FUNCTION "TE-ANEI" : VOID	// FC 78
AUTHOR : SIMATIC
FAMILY : EA_DIS
NAME : TE_ANEI
VERSION : 3.0
BEGIN
// (block stored without names or comments; labels and parameter names are numbered)
NETWORK
TITLE =
      L     #PARAM12;
      L     31;
      AW;
      T     MB 200;
      L     #PARAM4;
      T     MW 210;
      A     M 200.0;
      JC    M003;
      L     #PARAM3;
      T     MW 202;
      L     #PARAM1;
      L     W#16#4550;
      ==I;
      JC    M001;
      L     MB 203;
      SLW   3;
      LAR1;
      L     DBW [AR1,P#0.0];
      T     MW 204;
      JU    M002;
M001: NOP   0;
      L     MB 203;
      SLW   3;
      LAR1;
      L     DBW [AR1,P#0.0];
      T     MW 204;
M002: NOP   0;
M003: NOP   0;
NETWORK
TITLE =
      L     MW 210;
      L     2;
      ==I;
      JC    M004;
      JU    M007;
M004: A     M 200.0;
      JC    M008;
      L     MW 204;
      T     MW 240;
      AN    M 240.7;
      JC    M005;
      L     MW 240;
      NEGI;
      DTR;
      L     -1.000000e+00;
      *R;
      JU    M006;
M005: L     MW 240;
      DTR;
M006: T     MD 230;
      L     MD 230;
      L     1.000000e+01;
      /R;
      T     MD 238;
      L     MD 238;
      L     #PARAM7;
      -R;
      T     MD 218;
      L     #PARAM8;
      L     #PARAM7;
      -R;
      T     MD 242;
      L     MD 218;
      L     MD 242;
      /R;
      L     1.000000e+04;
      *R;
      T     MD 214;
      JU    M009;
M007: JU    M011;
M008: JU    M010;
M009: O(;
      L     MD 230;
      L     8.501000e+03;
      >=R;
      );
      O(;
      L     MD 230;
      L     1.000000e+04;
      >=R;
      );
      =     M 240.0;
      O(;
      L     -2.001000e+03;
      L     MD 230;
      >=R;
      );
      O(;
      L     -2.430000e+03;
      L     MD 230;
      >=R;
      );
      =     M 240.1;
      O(;
      L     -2.431000e+03;
      L     MD 230;
      >=R;
      );
      O(;
      L     -3.276800e+04;
      L     MD 230;
      >=R;
      );
      =     M 240.2;
      O(;
      L     MD 230;
      L     1.000000e+04;
      >=R;
      );
      O(;
      L     MD 230;
      L     3.276700e+04;
      >=R;
      );
      =     M 240.3;
      O(;
      L     MD 230;
      L     -2.000000e+03;
      >=R;
      );
      O(;
      L     MD 230;
      L     8.500000e+03;
      >=R;
      );
      =     M 240.4;
      O(;
      A     M 240.0;
      A     M 240.3;
      A     M 240.4;
      );
      O(;
      A     M 240.1;
      A     M 240.2;
      );
      =     M 200.6;
      A     M 200.3;
      A     M 200.6;
      =     M 200.7;
      L     MD 238;
      JU    M012;
M010: R     M 200.7;
      L     #PARAM6;
      T     MD 206;
      L     #PARAM7;
      -R;
      T     MD 244;
      L     #PARAM8;
      L     #PARAM7;
      -R;
      T     MD 248;
      L     MD 244;
      L     MD 248;
      /R;
      L     1.000000e+04;
      *R;
      T     MD 214;
      L     MD 206;
      JU    M014;
M011: JU    M015;
M012: AN    M 200.7;
      ON    M 200.1;
      JC    M013;
      JU    M014;
      L     1.000000e+04;
      T     MD 214;
      L     #PARAM8;
M013: AN    M 200.7;
      ON    M 200.2;
      JC    M014;
      L     0.000000e+00;
      T     MD 214;
      L     #PARAM7;
M014: T     #PARAM10;
      L     MD 214;
      T     #PARAM11;
      L     MB 200;
      T     #PARAM12;
M015: NOP   0;
NETWORK
TITLE =
      L     MW 210;
      L     4;
      ==I;
      JC    M016;
      JU    M020;
M016: A     M 200.0;
      JC    M021;
      L     MW 204;
      T     MW 240;
      AN    M 240.7;
      JC    M018;
M017: L     MW 240;
      NEGI;
      DTR;
      L     -1.000000e+00;
      *R;
      JU    M019;
M018: L     MW 240;
      L     32760;
      >I;
      JC    M017;
      L     MW 240;
      DTR;
M019: T     MD 230;
      L     2.764800e+04;
      /R;
      L     1.000000e+04;
      *R;
      T     MD 214;
      L     #PARAM8;
      L     #PARAM7;
      -R;
      L     1.000000e+04;
      /R;
      T     MD 218;
      L     MD 214;
      L     MD 218;
      *R;
      T     MD 234;
      L     #PARAM7;
      +R;
      T     MD 238;
      JU    M022;
M020: JU    M024;
M021: JU    M023;
M022: O(;
      L     MD 230;
      L     2.764900e+04;
      >=R;
      );
      O(;
      L     MD 230;
      L     3.251100e+04;
      >=R;
      );
      =     M 240.0;
      O(;
      L     -2.764900e+04;
      L     MD 230;
      >=R;
      );
      O(;
      L     -3.251200e+04;
      L     MD 230;
      >=R;
      );
      =     M 240.1;
      O(;
      L     -3.251300e+04;
      L     MD 230;
      >=R;
      );
      O(;
      L     -3.276800e+04;
      L     MD 230;
      >=R;
      );
      =     M 240.2;
      O(;
      L     MD 230;
      L     3.251200e+04;
      >=R;
      );
      O(;
      L     MD 230;
      L     3.276700e+04;
      >=R;
      );
      =     M 240.3;
      O(;
      L     MD 230;
      L     -2.764800e+04;
      >=R;
      );
      O(;
      L     MD 230;
      L     2.764800e+04;
      >=R;
      );
      =     M 240.4;
      O(;
      A     M 240.0;
      A     M 240.3;
      A     M 240.4;
      );
      O(;
      A     M 240.1;
      A     M 240.2;
      );
      =     M 200.6;
      A     M 200.3;
      A     M 200.6;
      =     M 200.7;
      L     MD 238;
      JU    M025;
M023: R     M 200.7;
      L     #PARAM6;
      T     MD 206;
      L     #PARAM7;
      -R;
      T     MD 244;
      L     #PARAM8;
      L     #PARAM7;
      -R;
      T     MD 248;
      L     MD 244;
      L     MD 248;
      /R;
      L     1.000000e+04;
      *R;
      T     MD 214;
      L     MD 206;
      JU    M027;
M024: JU    M028;
M025: AN    M 200.7;
      ON    M 200.1;
      JC    M026;
      JU    M027;
      L     1.000000e+04;
      T     MD 214;
      L     #PARAM8;
M026: AN    M 200.7;
      ON    M 200.2;
      JC    M027;
      L     0.000000e+00;
      T     MD 214;
      L     #PARAM7;
M027: T     #PARAM10;
      L     MD 214;
      T     #PARAM11;
      L     MB 200;
      T     #PARAM12;
M028: NOP   0;
NETWORK
TITLE =
      L     MW 210;
      L     6;
      ==I;
      JC    M029;
      JU    M033;
M029: A     M 200.0;
      JC    M034;
      L     MW 204;
      T     MW 240;
      AN    M 240.7;
      JC    M031;
M030: L     MW 240;
      NEGI;
      DTR;
      L     -1.000000e+00;
      *R;
      JU    M032;
M031: L     MW 240;
      L     32760;
      >I;
      JC    M030;
      L     MW 240;
      DTR;
M032: T     MD 230;
      L     2.764800e+04;
      /R;
      L     1.000000e+04;
      *R;
      T     MD 214;
      L     #PARAM8;
      L     #PARAM7;
      -R;
      L     1.000000e+04;
      /R;
      T     MD 218;
      L     MD 214;
      L     MD 218;
      *R;
      T     MD 234;
      L     #PARAM7;
      +R;
      T     MD 238;
      JU    M035;
M033: JU    M037;
M034: JU    M036;
M035: O(;
      L     MD 230;
      L     2.764900e+04;
      >=R;
      );
      O(;
      L     MD 230;
      L     3.251100e+04;
      >=R;
      );
      =     M 240.0;
      O(;
      L     -1.000000e+00;
      L     MD 230;
      >=R;
      );
      O(;
      L     -4.864000e+03;
      L     MD 230;
      >=R;
      );
      =     M 240.1;
      O(;
      L     -4.865000e+03;
      L     MD 230;
      >=R;
      );
      O(;
      L     -3.276800e+04;
      L     MD 230;
      >=R;
      );
      =     M 240.2;
      O(;
      L     MD 230;
      L     3.251200e+04;
      >=R;
      );
      O(;
      L     MD 230;
      L     3.276700e+04;
      >=R;
      );
      =     M 240.3;
      O(;
      L     MD 230;
      L     0.000000e+00;
      >=R;
      );
      O(;
      L     MD 230;
      L     2.764800e+04;
      >=R;
      );
      =     M 240.4;
      O(;
      A     M 240.0;
      A     M 240.3;
      A     M 240.4;
      );
      O(;
      A     M 240.1;
      A     M 240.2;
      );
      =     M 200.6;
      A     M 200.3;
      A     M 200.6;
      =     M 200.7;
      L     MD 238;
      JU    M038;
M036: R     M 200.7;
      L     #PARAM6;
      T     MD 206;
      L     #PARAM7;
      -R;
      T     MD 244;
      L     #PARAM8;
      L     #PARAM7;
      -R;
      T     MD 248;
      L     MD 244;
      L     MD 248;
      /R;
      L     1.000000e+04;
      *R;
      T     MD 214;
      L     MD 206;
      JU    M040;
M037: JU    M041;
M038: AN    M 200.7;
      ON    M 200.1;
      JC    M039;
      JU    M040;
      L     1.000000e+04;
      T     MD 214;
      L     #PARAM8;
M039: AN    M 200.7;
      ON    M 200.2;
      JC    M040;
      L     0.000000e+00;
      T     MD 214;
      L     #PARAM7;
M040: T     #PARAM10;
      L     MD 214;
      T     #PARAM11;
      L     MB 200;
      T     #PARAM12;
M041: NOP   0;
NETWORK
TITLE =
      L     MW 210;
      L     7;
      ==I;
      JC    M042;
      JU    M046;
M042: A     M 200.0;
      JC    M047;
      L     MW 204;
      T     MW 240;
      AN    M 240.7;
      JC    M044;
M043: L     MW 240;
      NEGI;
      DTR;
      L     -1.000000e+00;
      *R;
      JU    M045;
M044: L     MW 240;
      L     32760;
      >I;
      JC    M043;
      L     MW 240;
      DTR;
M045: T     MD 230;
      L     1.820000e+04;
      /R;
      L     1.000000e+04;
      *R;
      T     MD 214;
      L     #PARAM8;
      L     #PARAM7;
      -R;
      L     1.000000e+04;
      /R;
      T     MD 218;
      L     MD 214;
      L     MD 218;
      *R;
      T     MD 234;
      L     #PARAM7;
      +R;
      T     MD 238;
      JU    M048;
M046: JU    M050;
M047: JU    M049;
M048: O(;
      L     MD 230;
      L     1.820100e+04;
      >=R;
      );
      O(;
      L     MD 230;
      L     2.070000e+04;
      >=R;
      );
      =     M 240.0;
      O(;
      L     -1.000000e+00;
      L     MD 230;
      >=R;
      );
      O(;
      L     -1.200000e+03;
      L     MD 230;
      >=R;
      );
      =     M 240.1;
      L     -3.276800e+04;
      L     MD 230;
      >=R;
      =     M 240.2;
      L     MD 230;
      L     2.070100e+04;
      >=R;
      =     M 240.3;
      O(;
      L     MD 230;
      L     0.000000e+00;
      >=R;
      );
      O(;
      L     MD 230;
      L     1.820000e+04;
      >=R;
      );
      =     M 240.4;
      O(;
      A     M 240.0;
      A     M 240.3;
      A     M 240.4;
      );
      O(;
      A     M 240.1;
      A     M 240.2;
      );
      =     M 200.6;
      A     M 200.3;
      A     M 200.6;
      =     M 200.7;
      L     MD 238;
      JU    M051;
M049: R     M 200.7;
      L     #PARAM6;
      T     MD 206;
      L     #PARAM7;
      -R;
      T     MD 244;
      L     #PARAM8;
      L     #PARAM7;
      -R;
      T     MD 248;
      L     MD 244;
      L     MD 248;
      /R;
      L     1.000000e+04;
      *R;
      T     MD 214;
      L     MD 206;
      JU    M053;
M050: JU    M054;
M051: AN    M 200.7;
      ON    M 200.1;
      JC    M052;
      JU    M053;
      L     1.000000e+04;
      T     MD 214;
      L     #PARAM8;
M052: AN    M 200.7;
      ON    M 200.2;
      JC    M053;
      L     0.000000e+00;
      T     MD 214;
      L     #PARAM7;
M053: T     #PARAM10;
      L     MD 214;
      T     #PARAM11;
      L     MB 200;
      T     #PARAM12;
M054: NOP   0;
NETWORK
TITLE =
      L     MW 210;
      L     8;
      ==I;
      JC    M055;
      JU    M059;
M055: A     M 200.0;
      JC    M060;
      L     MW 204;
      T     MW 240;
      AN    M 240.7;
      JC    M057;
M056: L     MW 240;
      NEGI;
      DTR;
      L     -1.000000e+00;
      *R;
      JU    M058;
M057: L     MW 240;
      L     32760;
      >I;
      JC    M056;
      L     MW 240;
      DTR;
M058: T     MD 230;
      L     2.315000e+04;
      /R;
      L     1.000000e+04;
      *R;
      T     MD 214;
      L     #PARAM8;
      L     #PARAM7;
      -R;
      L     1.000000e+04;
      /R;
      T     MD 218;
      L     MD 214;
      L     MD 218;
      *R;
      T     MD 234;
      L     #PARAM7;
      +R;
      T     MD 238;
      JU    M061;
M059: JU    M063;
M060: JU    M062;
M061: O(;
      L     MD 230;
      L     2.500000e+04;
      >=R;
      );
      O(;
      L     MD 230;
      L     2.315100e+04;
      >=R;
      );
      =     M 240.0;
      O(;
      L     -1.000000e+00;
      L     MD 230;
      >=R;
      );
      O(;
      L     -1.200000e+03;
      L     MD 230;
      >=R;
      );
      =     M 240.1;
      L     -3.276800e+04;
      L     MD 230;
      >=R;
      =     M 240.2;
      L     MD 230;
      L     2.500100e+04;
      >=R;
      =     M 240.3;
      O(;
      L     MD 230;
      L     0.000000e+00;
      >=R;
      );
      O(;
      L     MD 230;
      L     2.315000e+04;
      >=R;
      );
      =     M 240.4;
      O(;
      A     M 240.0;
      A     M 240.3;
      A     M 240.4;
      );
      O(;
      A     M 240.1;
      A     M 240.2;
      );
      =     M 200.6;
      A     M 200.3;
      A     M 200.6;
      =     M 200.7;
      L     MD 238;
      JU    M064;
M062: R     M 200.7;
      L     #PARAM6;
      T     MD 206;
      L     #PARAM7;
      -R;
      T     MD 244;
      L     #PARAM8;
      L     #PARAM7;
      -R;
      T     MD 248;
      L     MD 244;
      L     MD 248;
      /R;
      L     1.000000e+04;
      *R;
      T     MD 214;
      L     MD 206;
      JU    M066;
M063: JU    M067;
M064: AN    M 200.7;
      ON    M 200.1;
      JC    M065;
      JU    M066;
      L     1.000000e+04;
      T     MD 214;
      L     #PARAM8;
M065: AN    M 200.7;
      ON    M 200.2;
      JC    M066;
      L     0.000000e+00;
      T     MD 214;
      L     #PARAM7;
M066: T     #PARAM10;
      L     MD 214;
      T     #PARAM11;
      L     MB 200;
      T     #PARAM12;
M067: NOP   0;
NETWORK
TITLE =
      L     MW 210;
      L     9;
      ==I;
      JC    M068;
      JU    M073;
M068: A     M 200.0;
      JC    M074;
      L     MW 204;
      T     MW 240;
      AN    M 240.7;
      JC    M070;
M069: L     MW 240;
      NEGI;
      DTR;
      L     -1.000000e+00;
      *R;
      JU    M071;
M070: L     MW 240;
      L     32760;
      >I;
      JC    M069;
      L     MW 240;
      DTR;
      JU    M072;
M071: T     MD 230;
      L     #PARAM7;
      L     1.000000e+01;
      *R;
      T     MD 242;
      L     MD 230;
      L     MD 242;
      -R;
      L     1.270000e+04;
      /R;
      L     1.000000e+04;
      *R;
      T     MD 214;
      L     #PARAM8;
      L     #PARAM7;
      -R;
      L     1.000000e+04;
      /R;
      T     MD 218;
      L     MD 214;
      L     MD 218;
      *R;
      T     MD 234;
      L     #PARAM7;
      +R;
      T     MD 238;
      JU    M075;
M072: T     MD 230;
      L     #PARAM7;
      L     -1.000000e+01;
      *R;
      T     MD 242;
      L     MD 230;
      L     MD 242;
      +R;
      L     1.270000e+04;
      /R;
      L     1.000000e+04;
      *R;
      T     MD 214;
      L     #PARAM8;
      L     #PARAM7;
      -R;
      L     1.000000e+04;
      /R;
      T     MD 218;
      L     MD 214;
      L     MD 218;
      *R;
      T     MD 234;
      L     #PARAM7;
      +R;
      T     MD 238;
      JU    M075;
M073: JU    M077;
M074: JU    M076;
M075: O(;
      L     MD 230;
      L     1.200000e+04;
      >=R;
      );
      O(;
      L     MD 230;
      L     1.000100e+04;
      >=R;
      );
      =     M 240.0;
      O(;
      L     -1.000000e+00;
      L     MD 230;
      >=R;
      );
      O(;
      L     -1.200000e+03;
      L     MD 230;
      >=R;
      );
      =     M 240.1;
      L     -3.276800e+04;
      L     MD 230;
      >=R;
      =     M 240.2;
      L     MD 230;
      L     2.500100e+04;
      >=R;
      =     M 240.3;
      O(;
      L     MD 230;
      L     -2.700000e+03;
      >=R;
      );
      O(;
      L     MD 230;
      L     1.000000e+04;
      >=R;
      );
      =     M 240.4;
      O(;
      A     M 240.0;
      A     M 240.3;
      A     M 240.4;
      );
      O(;
      A     M 240.1;
      A     M 240.2;
      );
      =     M 200.6;
      A     M 200.3;
      A     M 200.6;
      =     M 200.7;
      L     MD 238;
      JU    M078;
M076: R     M 200.7;
      L     #PARAM6;
      T     MD 206;
      L     #PARAM7;
      -R;
      T     MD 244;
      L     #PARAM8;
      L     #PARAM7;
      -R;
      T     MD 248;
      L     MD 244;
      L     MD 248;
      /R;
      L     1.000000e+04;
      *R;
      T     MD 214;
      L     MD 206;
      JU    M080;
M077: JU    M081;
M078: AN    M 200.7;
      ON    M 200.1;
      JC    M079;
      JU    M080;
      L     1.000000e+04;
      T     MD 214;
      L     #PARAM8;
M079: AN    M 200.7;
      ON    M 200.2;
      JC    M040;
      L     0.000000e+00;
      T     MD 214;
      L     #PARAM7;
M080: T     #PARAM10;
      L     MD 214;
      T     #PARAM11;
      L     MB 200;
      T     #PARAM12;
M081: NOP   0;
NETWORK
TITLE =
      L     MW 210;
      L     10;
      ==I;
      JC    M082;
      JU    M085;
M082: A     M 200.0;
      JC    M086;
      L     MW 204;
      T     MW 240;
      AN    M 240.7;
      JC    M083;
      L     MW 240;
      NEGI;
      DTR;
      L     -1.000000e+00;
      *R;
      JU    M084;
M083: L     MW 240;
      DTR;
M084: T     MD 230;
      L     MD 230;
      L     1.000000e+01;
      /R;
      T     MD 238;
      L     MD 238;
      L     #PARAM7;
      -R;
      T     MD 218;
      L     #PARAM8;
      L     #PARAM7;
      -R;
      T     MD 242;
      L     MD 218;
      L     MD 242;
      /R;
      L     1.000000e+04;
      *R;
      T     MD 214;
      JU    M087;
M085: JU    M089;
M086: JU    M088;
M087: O(;
      L     MD 230;
      L     1.200100e+04;
      >=R;
      );
      O(;
      L     MD 230;
      L     1.450000e+04;
      >=R;
      );
      =     M 240.0;
      L     -2.100000e+03;
      L     MD 230;
      >=R;
      =     M 240.1;
      L     -2.100000e+03;
      L     MD 230;
      >=R;
      =     M 240.2;
      L     MD 230;
      L     1.450100e+04;
      >=R;
      =     M 240.3;
      O(;
      L     MD 230;
      L     -2.100000e+03;
      >=R;
      );
      O(;
      L     MD 230;
      L     1.200000e+03;
      >=R;
      );
      =     M 240.4;
      O(;
      A     M 240.0;
      A     M 240.3;
      A     M 240.4;
      );
      O(;
      A     M 240.1;
      A     M 240.2;
      );
      =     M 200.6;
      A     M 200.3;
      A     M 200.6;
      =     M 200.7;
      L     MD 238;
      JU    M090;
M088: R     M 200.7;
      L     #PARAM6;
      T     MD 206;
      L     #PARAM7;
      -R;
      T     MD 244;
      L     #PARAM8;
      L     #PARAM7;
      -R;
      T     MD 248;
      L     MD 244;
      L     MD 248;
      /R;
      L     1.000000e+04;
      *R;
      T     MD 214;
      L     MD 206;
      JU    M092;
M089: JU    M093;
M090: AN    M 200.7;
      ON    M 200.1;
      JC    M091;
      JU    M092;
      L     1.000000e+04;
      T     MD 214;
      L     #PARAM8;
M091: AN    M 200.7;
      ON    M 200.2;
      JC    M092;
      L     0.000000e+00;
      T     MD 214;
      L     #PARAM7;
M092: T     #PARAM10;
      L     MD 214;
      T     #PARAM11;
      L     MB 200;
      T     #PARAM12;
M093: NOP   0;
NETWORK
TITLE =
      L     MW 210;
      L     11;
      ==I;
      JC    M094;
      JU    M097;
M094: A     M 200.0;
      JC    M098;
      L     MW 204;
      T     MW 240;
      AN    M 240.7;
      JC    M095;
      L     MW 240;
      NEGI;
      DTR;
      L     -1.000000e+00;
      *R;
      JU    M096;
M095: L     MW 240;
      DTR;
M096: T     MD 230;
      L     MD 230;
      L     1.000000e+01;
      /R;
      T     MD 238;
      L     MD 238;
      L     #PARAM7;
      -R;
      T     MD 218;
      L     #PARAM8;
      L     #PARAM7;
      -R;
      T     MD 242;
      L     MD 218;
      L     MD 242;
      /R;
      L     1.000000e+04;
      *R;
      T     MD 214;
      JU    M099;
M097: JU    M101;
M098: JU    M100;
M099: O(;
      L     MD 230;
      L     1.666200e+04;
      >=R;
      );
      O(;
      L     MD 230;
      L     1.372100e+04;
      >=R;
      );
      =     M 240.0;
      L     -2.700000e+03;
      L     MD 230;
      >=R;
      =     M 240.1;
      L     -2.700000e+03;
      L     MD 230;
      >=R;
      =     M 240.2;
      L     MD 230;
      L     1.622100e+04;
      >=R;
      =     M 240.3;
      O(;
      L     MD 230;
      L     -2.700000e+03;
      >=R;
      );
      O(;
      L     MD 230;
      L     1.372000e+03;
      >=R;
      );
      =     M 240.4;
      O(;
      A     M 240.0;
      A     M 240.3;
      A     M 240.4;
      );
      O(;
      A     M 240.1;
      A     M 240.2;
      );
      =     M 200.6;
      A     M 200.3;
      A     M 200.6;
      =     M 200.7;
      L     MD 238;
      JU    M102;
M100: R     M 200.7;
      L     #PARAM6;
      T     MD 206;
      L     #PARAM7;
      -R;
      T     MD 244;
      L     #PARAM8;
      L     #PARAM7;
      -R;
      T     MD 248;
      L     MD 244;
      L     MD 248;
      /R;
      L     1.000000e+04;
      *R;
      T     MD 214;
      L     MD 206;
      JU    M104;
M101: JU    M105;
M102: AN    M 200.7;
      ON    M 200.1;
      JC    M103;
      JU    M104;
      L     1.000000e+04;
      T     MD 214;
      L     #PARAM8;
M103: AN    M 200.7;
      ON    M 200.2;
      JC    M104;
      L     0.000000e+00;
      T     MD 214;
      L     #PARAM7;
M104: T     #PARAM10;
      L     MD 214;
      T     #PARAM11;
      L     MB 200;
      T     #PARAM12;
M105: NOP   0;
NETWORK
TITLE =
      L     MW 210;
      L     12;
      ==I;
      JC    M106;
      JU    M109;
M106: A     M 200.0;
      JC    M110;
      L     MW 204;
      T     MW 240;
      AN    M 240.7;
      JC    M107;
      L     MW 240;
      NEGI;
      DTR;
      L     -1.000000e+00;
      *R;
      JU    M108;
M107: L     MW 240;
      DTR;
M108: T     MD 230;
      L     MD 230;
      L     1.000000e+01;
      /R;
      T     MD 238;
      L     MD 238;
      L     #PARAM7;
      -R;
      T     MD 218;
      L     #PARAM8;
      L     #PARAM7;
      -R;
      T     MD 242;
      L     MD 218;
      L     MD 242;
      /R;
      L     1.000000e+04;
      *R;
      T     MD 214;
      JU    M111;
M109: JU    M113;
M110: JU    M112;
M111: O(;
      L     MD 230;
      L     1.150000e+04;
      >=R;
      );
      O(;
      L     MD 230;
      L     9.001000e+03;
      >=R;
      );
      =     M 240.0;
      L     -2.000000e+03;
      L     MD 230;
      >=R;
      =     M 240.1;
      L     -2.000000e+03;
      L     MD 230;
      >=R;
      =     M 240.2;
      L     MD 230;
      L     9.001000e+03;
      >=R;
      =     M 240.3;
      O(;
      L     MD 230;
      L     -2.000000e+03;
      >=R;
      );
      O(;
      L     MD 230;
      L     9.000000e+03;
      >=R;
      );
      =     M 240.4;
      O(;
      A     M 240.0;
      A     M 240.3;
      A     M 240.4;
      );
      O(;
      A     M 240.1;
      A     M 240.2;
      );
      =     M 200.6;
      A     M 200.3;
      A     M 200.6;
      =     M 200.7;
      L     MD 238;
      JU    M114;
M112: R     M 200.7;
      L     #PARAM6;
      T     MD 206;
      L     #PARAM7;
      -R;
      T     MD 244;
      L     #PARAM8;
      L     #PARAM7;
      -R;
      T     MD 248;
      L     MD 244;
      L     MD 248;
      /R;
      L     1.000000e+04;
      *R;
      T     MD 214;
      L     MD 206;
      JU    M116;
M113: JU    M117;
M114: AN    M 200.7;
      ON    M 200.1;
      JC    M115;
      JU    M116;
      L     1.000000e+04;
      T     MD 214;
      L     #PARAM8;
M115: AN    M 200.7;
      ON    M 200.2;
      JC    M116;
      L     0.000000e+00;
      T     MD 214;
      L     #PARAM7;
M116: T     #PARAM10;
      L     MD 214;
      T     #PARAM11;
      L     MB 200;
      T     #PARAM12;
M117: NOP   0;
NETWORK
TITLE =
      L     MW 210;
      L     12;
      ==I;
      JC    M118;
      JU    M121;
M118: A     M 200.0;
      JC    M122;
      L     MW 204;
      T     MW 240;
      AN    M 240.7;
      JC    M119;
      L     MW 240;
      NEGI;
      DTR;
      L     -1.000000e+00;
      *R;
      JU    M120;
M119: L     MW 240;
      DTR;
M120: T     MD 230;
      L     MD 230;
      L     1.000000e+01;
      /R;
      T     MD 238;
      L     MD 238;
      L     #PARAM7;
      -R;
      T     MD 218;
      L     #PARAM8;
      L     #PARAM7;
      -R;
      T     MD 242;
      L     MD 218;
      L     MD 242;
      /R;
      L     1.000000e+04;
      *R;
      T     MD 214;
      JU    M123;
M121: JU    M125;
M122: JU    M124;
M123: O(;
      L     MD 230;
      L     1.550000e+04;
      >=R;
      );
      O(;
      L     MD 230;
      L     1.300100e+04;
      >=R;
      );
      =     M 240.0;
      L     -2.700000e+03;
      L     MD 230;
      >=R;
      =     M 240.1;
      L     -2.700000e+03;
      L     MD 230;
      >=R;
      =     M 240.2;
      L     MD 230;
      L     1.550100e+04;
      >=R;
      =     M 240.3;
      O(;
      L     MD 230;
      L     -2.700000e+03;
      >=R;
      );
      O(;
      L     MD 230;
      L     1.550000e+03;
      >=R;
      );
      =     M 240.4;
      O(;
      A     M 240.0;
      A     M 240.3;
      A     M 240.4;
      );
      O(;
      A     M 240.1;
      A     M 240.2;
      );
      =     M 200.6;
      A     M 200.3;
      A     M 200.6;
      =     M 200.7;
      L     MD 238;
      JU    M126;
M124: R     M 200.7;
      L     #PARAM6;
      T     MD 206;
      L     #PARAM7;
      -R;
      T     MD 244;
      L     #PARAM8;
      L     #PARAM7;
      -R;
      T     MD 248;
      L     MD 244;
      L     MD 248;
      /R;
      L     1.000000e+04;
      *R;
      T     MD 214;
      L     MD 206;
      JU    M128;
M125: JU    M129;
M126: AN    M 200.7;
      ON    M 200.1;
      JC    M127;
      JU    M128;
      L     1.000000e+04;
      T     MD 214;
      L     #PARAM8;
M127: AN    M 200.7;
      ON    M 200.2;
      JC    M128;
      L     0.000000e+00;
      T     MD 214;
      L     #PARAM7;
M128: T     #PARAM10;
      L     MD 214;
      T     #PARAM11;
      L     MB 200;
      T     #PARAM12;
M129: NOP   0;
NETWORK
TITLE =
      L     MW 210;
      L     14;
      ==I;
      JC    M130;
      JU    M133;
M130: A     M 200.0;
      JC    M134;
      L     MW 204;
      T     MW 240;
      AN    M 240.7;
      JC    M131;
      L     MW 240;
      NEGI;
      DTR;
      L     -1.000000e+00;
      *R;
      JU    M132;
M131: L     MW 240;
      DTR;
M132: T     MD 230;
      L     MD 230;
      L     1.000000e+01;
      /R;
      T     MD 238;
      L     MD 238;
      L     #PARAM7;
      -R;
      T     MD 218;
      L     #PARAM8;
      L     #PARAM7;
      -R;
      T     MD 242;
      L     MD 218;
      L     MD 242;
      /R;
      L     1.000000e+04;
      *R;
      T     MD 214;
      JU    M135;
M133: JU    M137;
M134: JU    M136;
M135: O(;
      L     MD 230;
      L     2.019000e+04;
      >=R;
      );
      O(;
      L     MD 230;
      L     1.769100e+04;
      >=R;
      );
      =     M 240.0;
      O(;
      L     -5.010000e+02;
      L     MD 230;
      >=R;
      );
      O(;
      L     -1.700000e+03;
      L     MD 230;
      >=R;
      );
      =     M 240.1;
      O(;
      L     2.090100e+04;
      L     MD 230;
      >=R;
      );
      O(;
      L     -1.200000e+03;
      L     MD 230;
      >=R;
      );
      =     M 240.2;
      O(;
      L     -1.000000e+00;
      L     MD 230;
      >=R;
      );
      O(;
      L     -1.200000e+03;
      L     MD 230;
      >=R;
      );
      =     M 240.3;
      O(;
      L     MD 230;
      L     -5.000000e+02;
      >=R;
      );
      O(;
      L     MD 230;
      L     1.769000e+04;
      >=R;
      );
      =     M 240.4;
      O(;
      A     M 240.0;
      A     M 240.3;
      A     M 240.4;
      );
      O(;
      A     M 240.1;
      A     M 240.2;
      );
      =     M 200.6;
      A     M 200.3;
      A     M 200.6;
      =     M 200.7;
      L     MD 238;
      JU    M138;
M136: R     M 200.7;
      L     #PARAM6;
      T     MD 206;
      L     #PARAM7;
      -R;
      T     MD 244;
      L     #PARAM8;
      L     #PARAM7;
      -R;
      T     MD 248;
      L     MD 244;
      L     MD 248;
      /R;
      L     1.000000e+04;
      *R;
      T     MD 214;
      L     MD 206;
      JU    M140;
M137: JU    M141;
M138: AN    M 200.7;
      ON    M 200.1;
      JC    M139;
      JU    M140;
      L     1.000000e+04;
      T     MD 214;
      L     #PARAM8;
M139: AN    M 200.7;
      ON    M 200.2;
      JC    M140;
      L     0.000000e+00;
      T     MD 214;
      L     #PARAM7;
M140: T     #PARAM10;
      L     MD 214;
      T     #PARAM11;
      L     MB 200;
      T     #PARAM12;
M141: NOP   0;
NETWORK
TITLE =
      L     MW 210;
      L     14;
      ==I;
      JC    M142;
      JU    M145;
M142: A     M 200.0;
      JC    M146;
      L     MW 204;
      T     MW 240;
      AN    M 240.7;
      JC    M143;
      L     MW 240;
      NEGI;
      DTR;
      L     -1.000000e+00;
      *R;
      JU    M144;
M143: L     MW 240;
      DTR;
M144: T     MD 230;
      L     MD 230;
      L     1.000000e+01;
      /R;
      T     MD 238;
      L     MD 238;
      L     #PARAM7;
      -R;
      T     MD 218;
      L     #PARAM8;
      L     #PARAM7;
      -R;
      T     MD 242;
      L     MD 218;
      L     MD 242;
      /R;
      L     1.000000e+04;
      *R;
      T     MD 214;
      JU    M147;
M145: JU    M149;
M146: JU    M148;
M147: O(;
      L     MD 230;
      L     1.666200e+04;
      >=R;
      );
      O(;
      L     MD 230;
      L     1.372100e+04;
      >=R;
      );
      =     M 240.0;
      L     -2.700000e+03;
      L     MD 230;
      >=R;
      =     M 240.1;
      L     -2.700000e+03;
      L     MD 230;
      >=R;
      =     M 240.2;
      L     MD 230;
      L     1.622100e+04;
      >=R;
      =     M 240.3;
      O(;
      L     MD 230;
      L     -2.700000e+03;
      >=R;
      );
      O(;
      L     MD 230;
      L     1.372000e+03;
      >=R;
      );
      =     M 240.4;
      O(;
      A     M 240.0;
      A     M 240.3;
      A     M 240.4;
      );
      O(;
      A     M 240.1;
      A     M 240.2;
      );
      =     M 200.6;
      A     M 200.3;
      A     M 200.6;
      =     M 200.7;
      L     MD 238;
      JU    M150;
M148: R     M 200.7;
      L     #PARAM6;
      T     MD 206;
      L     #PARAM7;
      -R;
      T     MD 244;
      L     #PARAM8;
      L     #PARAM7;
      -R;
      T     MD 248;
      L     MD 244;
      L     MD 248;
      /R;
      L     1.000000e+04;
      *R;
      T     MD 214;
      L     MD 206;
      JU    M152;
M149: JU    M153;
M150: AN    M 200.7;
      ON    M 200.1;
      JC    M151;
      JU    M152;
      L     1.000000e+04;
      T     MD 214;
      L     #PARAM8;
M151: AN    M 200.7;
      ON    M 200.2;
      JC    M152;
      L     0.000000e+00;
      T     MD 214;
      L     #PARAM7;
M152: T     #PARAM10;
      L     MD 214;
      T     #PARAM11;
      L     MB 200;
      T     #PARAM12;
M153: NOP   0;
NETWORK
TITLE =
      L     0;
      L     #PARAM9;
      ==I;
      BEC;
      T     MW 206;
      T     MW 220;
      L     MB 206;
      SLW   3;
      LAR1;
      L     DBW [AR1,P#0.0];
      T     MW 208;
      L     MW 220;
      SLW   12;
      SRW   12;
      T     MW 220;
      L     8;
      L     MB 221;
      >I;
      JC    M154;
      +     -8;
      SLW   8;
      INC   208;
      JU    M155;
M154: SLW   8;
      INC   209;
M155: T     MW 210;
      L     MB 210;
      L     MB 211;
      SLW   3;
      OW;
      LAR2;
      A     M 200.7;
      =     M [AR2,P#0.0];
      L     MB 206;
      SLW   3;
      LAR1;
      L     MW 208;
      T     DBW [AR1,P#0.0];
END_FUNCTION

FUNCTION "TE-ANAU" : VOID	// FC 79
AUTHOR : SIMATIC
FAMILY : EA_DIS
NAME : TE_ANAU
VERSION : 3.0
BEGIN
// (block stored without names or comments; labels and parameter names are numbered)
NETWORK
TITLE =
      L     #PARAM1;
      T     MB 255;
      L     #PARAM3;
      T     MB 254;
      L     1;
      >I;
      JC    M001;
      L     #PARAM2;
      L     2.764800e+00;
      *R;
      RND;
      T     MW 240;
      JU    M004;
M001: L     #PARAM2;
      L     0.000000e+00;
      <R;
      JC    M002;
      TAK;
      L     2.764800e+00;
      *R;
      T     MD 250;
      JU    M003;
M002: TAK;
      L     -1.000000e+00;
      *R;
M003: RND;
      T     MW 240;
M004: A     M 255.1;
      JC    M005;
      L     MW 240;
      T     #PARAM4;
M005: NOP   0;
END_FUNCTION

FUNCTION "FC 110" : VOID	// FC 110
VERSION : 0.1
BEGIN
// (block stored without names or comments; labels and parameter names are numbered)
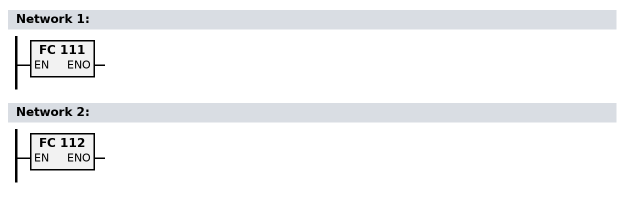
NETWORK
TITLE =
      CALL  "FC 111";
      NOP   0;
NETWORK
TITLE =
      CALL  "FC 112";
      NOP   0;
END_FUNCTION

FUNCTION "FC 111" : VOID	// FC 111
VERSION : 0.1
BEGIN
// (block stored without names or comments; labels and parameter names are numbered)
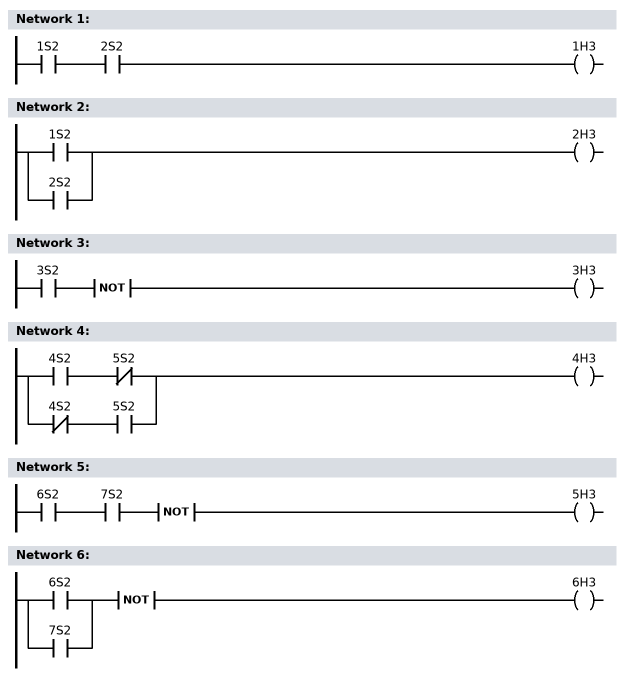
NETWORK
TITLE =
      A     "1S2";
      A     "2S2";
      =     "1H3";
NETWORK
TITLE =
      O     "1S2";
      O     "2S2";
      =     "2H3";
NETWORK
TITLE =
      A     "3S2";
      NOT;
      =     "3H3";
NETWORK
TITLE =
      A     "4S2";
      AN    "5S2";
      O;
      AN    "4S2";
      A     "5S2";
      =     "4H3";
NETWORK
TITLE =
      A     "6S2";
      A     "7S2";
      NOT;
      =     "5H3";
NETWORK
TITLE =
      A(;
      O     "6S2";
      O     "7S2";
      );
      NOT;
      =     "6H3";
END_FUNCTION

FUNCTION "FC 112" : VOID	// FC 112
VERSION : 0.1
BEGIN
// (block stored without names or comments; labels and parameter names are numbered)
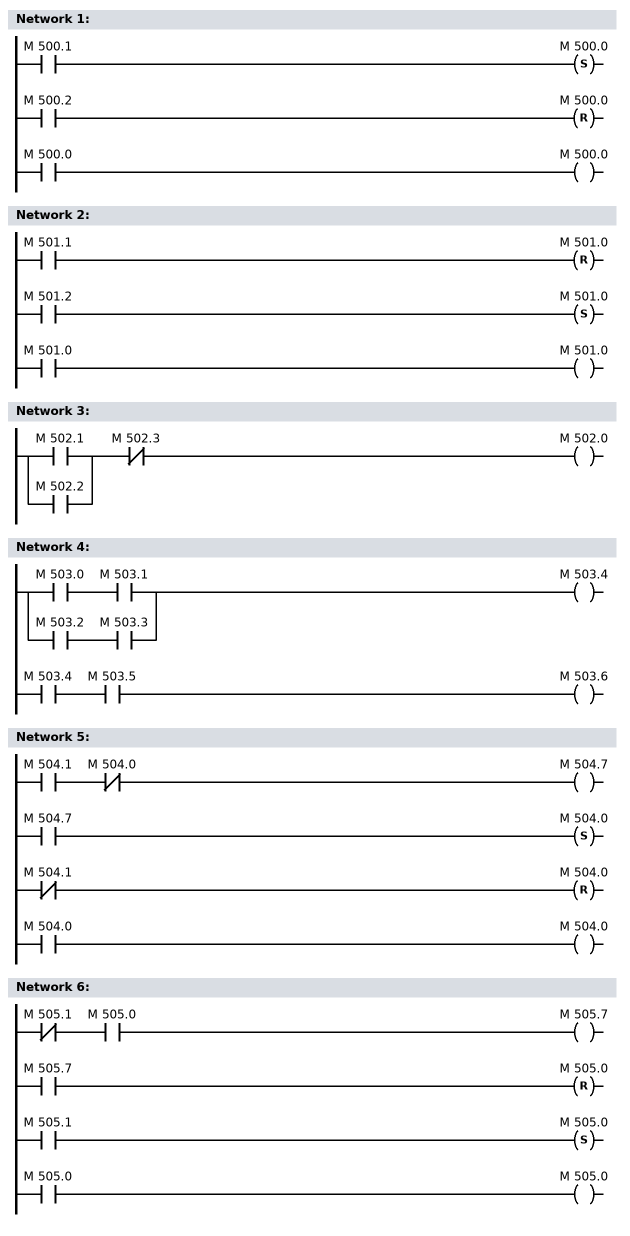
NETWORK
TITLE =
      A     M 500.1;
      S     M 500.0;
      A     M 500.2;
      R     M 500.0;
      A     M 500.0;
      =     M 500.0;
NETWORK
TITLE =
      A     M 501.1;
      R     M 501.0;
      A     M 501.2;
      S     M 501.0;
      A     M 501.0;
      =     M 501.0;
NETWORK
TITLE =
      A(;
      O     M 502.1;
      O     M 502.2;
      );
      AN    M 502.3;
      =     M 502.0;
NETWORK
TITLE =
      A(;
      A     M 503.0;
      A     M 503.1;
      O;
      A     M 503.2;
      A     M 503.3;
      );
      =     M 503.4;
      A     M 503.4;
      A     M 503.5;
      =     M 503.6;
NETWORK
TITLE =
      A     M 504.1;
      AN    M 504.0;
      =     M 504.7;
      A     M 504.7;
      S     M 504.0;
      AN    M 504.1;
      R     M 504.0;
      A     M 504.0;
      =     M 504.0;
NETWORK
TITLE =
      AN    M 505.1;
      A     M 505.0;
      =     M 505.7;
      A     M 505.7;
      R     M 505.0;
      A     M 505.1;
      S     M 505.0;
      A     M 505.0;
      =     M 505.0;
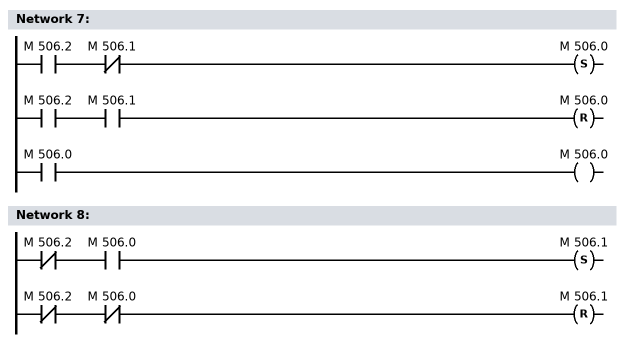
NETWORK
TITLE =
      A     M 506.2;
      AN    M 506.1;
      S     M 506.0;
      A     M 506.2;
      A     M 506.1;
      R     M 506.0;
      A     M 506.0;
      =     M 506.0;
NETWORK
TITLE =
      AN    M 506.2;
      A     M 506.0;
      S     M 506.1;
      AN    M 506.2;
      AN    M 506.0;
      R     M 506.1;
      NOP   0;
END_FUNCTION

FUNCTION "FC 113" : VOID	// FC 113
VERSION : 0.1
BEGIN
// (block stored without names or comments; labels and parameter names are numbered)
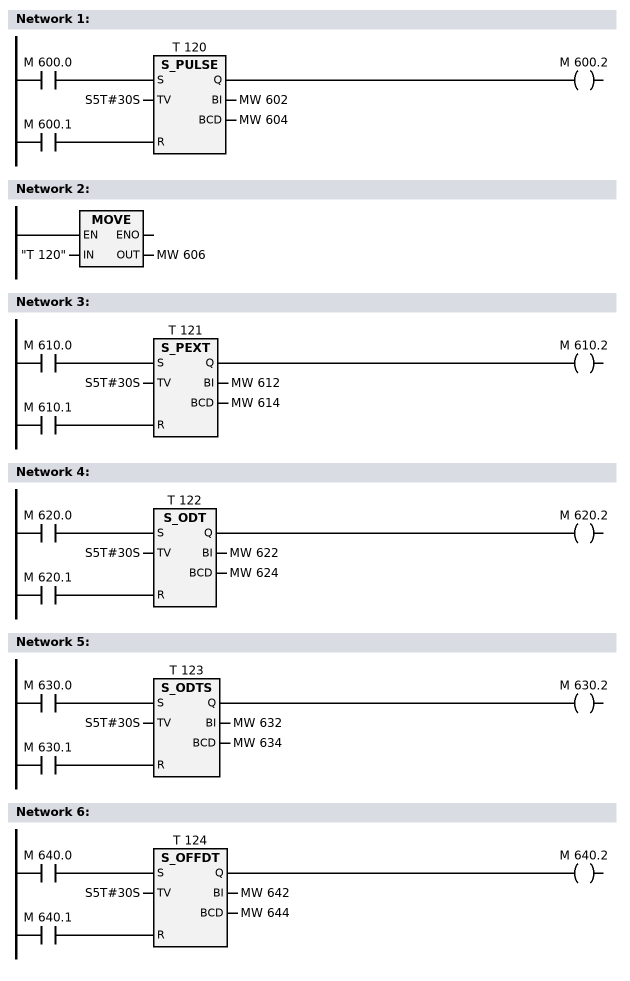
NETWORK
TITLE =
      A     M 600.0;
      L     S5T#30S;
      SP    "T 120";
      A     M 600.1;
      R     "T 120";
      L     "T 120";
      T     MW 602;
      LC    "T 120";
      T     MW 604;
      A     "T 120";
      =     M 600.2;
NETWORK
TITLE =
      L     "T 120";
      T     MW 606;
      NOP   0;
NETWORK
TITLE =
      A     M 610.0;
      L     S5T#30S;
      SE    "T 121";
      A     M 610.1;
      R     "T 121";
      L     "T 121";
      T     MW 612;
      LC    "T 121";
      T     MW 614;
      A     "T 121";
      =     M 610.2;
NETWORK
TITLE =
      A     M 620.0;
      L     S5T#30S;
      SD    "T 122";
      A     M 620.1;
      R     "T 122";
      L     "T 122";
      T     MW 622;
      LC    "T 122";
      T     MW 624;
      A     "T 122";
      =     M 620.2;
NETWORK
TITLE =
      A     M 630.0;
      L     S5T#30S;
      SS    "T 123";
      A     M 630.1;
      R     "T 123";
      L     "T 123";
      T     MW 632;
      LC    "T 123";
      T     MW 634;
      A     "T 123";
      =     M 630.2;
NETWORK
TITLE =
      A     M 640.0;
      L     S5T#30S;
      SF    "T 124";
      A     M 640.1;
      R     "T 124";
      L     "T 124";
      T     MW 642;
      LC    "T 124";
      T     MW 644;
      A     "T 124";
      =     M 640.2;
END_FUNCTION

FUNCTION "FC 114" : VOID	// FC 114
VERSION : 0.1
BEGIN
// (block stored without names or comments; labels and parameter names are numbered)
NETWORK
TITLE =
      A     M 700.0;
      CU    "Z 120";
      A     M 700.1;
      CD    "Z 120";
      A     M 700.2;
      L     MW 702;
      S     "Z 120";
      A     M 700.3;
      R     "Z 120";
      L     "Z 120";
      T     MW 704;
      LC    "Z 120";
      T     MW 706;
      A     "Z 120";
      =     M 700.4;
NETWORK
TITLE =
      A     M 710.0;
      CU    "Z 121";
      BLD   101;
      A     M 710.2;
      L     MW 712;
      S     "Z 121";
      A     M 710.3;
      R     "Z 121";
      L     "Z 121";
      T     MW 714;
      LC    "Z 121";
      T     MW 716;
      A     "Z 121";
      =     M 710.4;
NETWORK
TITLE =
      A     M 720.0;
      CD    "Z 122";
      BLD   101;
      A     M 720.2;
      L     MW 722;
      S     "Z 122";
      A     M 720.3;
      R     "Z 122";
      L     "Z 122";
      T     MW 724;
      LC    "Z 122";
      T     MW 726;
      A     "Z 122";
      =     M 720.4;
END_FUNCTION

FUNCTION "FC 120" : VOID	// FC 120
VERSION : 0.1
BEGIN
// (block stored without names or comments; labels and parameter names are numbered)
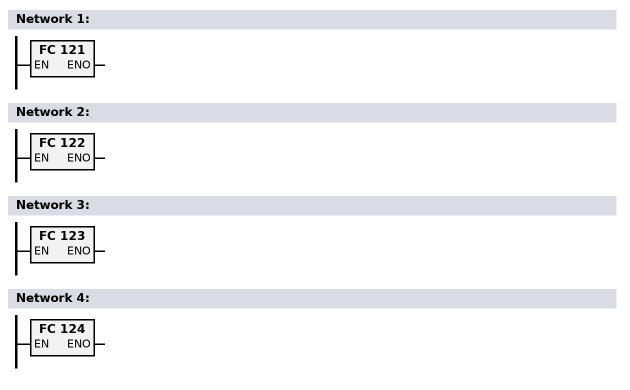
NETWORK
TITLE =
      CALL  "FC 121";
      NOP   0;
NETWORK
TITLE =
      CALL  "FC 122";
      NOP   0;
NETWORK
TITLE =
      CALL  "FC 123";
      NOP   0;
NETWORK
TITLE =
      CALL  "FC 124";
      NOP   0;
END_FUNCTION

FUNCTION "FC 121" : VOID	// FC 121
VERSION : 0.1
BEGIN
// (block stored without names or comments; labels and parameter names are numbered)
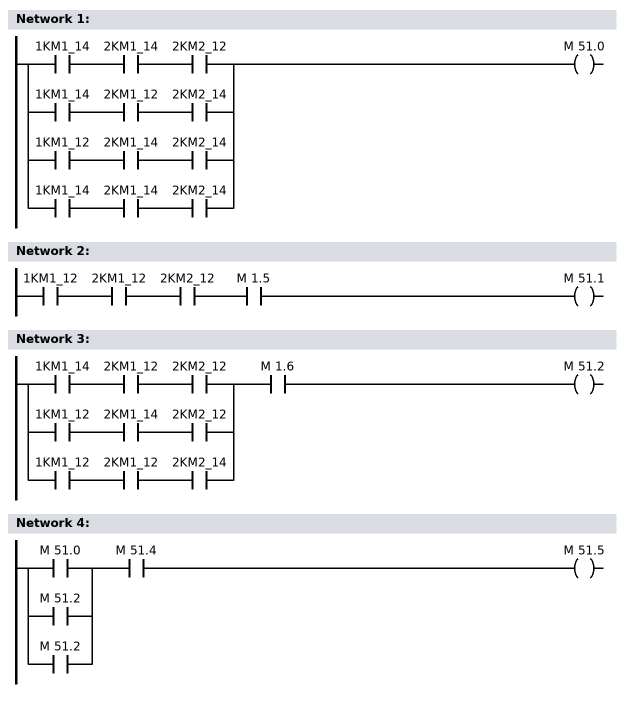
NETWORK
TITLE =
      A     "1KM1_14";
      A     "2KM1_14";
      A     "2KM2_12";
      O;
      A     "1KM1_14";
      A     "2KM1_12";
      A     "2KM2_14";
      O;
      A     "1KM1_12";
      A     "2KM1_14";
      A     "2KM2_14";
      O;
      A     "1KM1_14";
      A     "2KM1_14";
      A     "2KM2_14";
      =     "M 51.0";
NETWORK
TITLE =
      A     "1KM1_12";
      A     "2KM1_12";
      A     "2KM2_12";
      A     "M 1.5";
      =     "M 51.1";
NETWORK
TITLE =
      A(;
      A     "1KM1_14";
      A     "2KM1_12";
      A     "2KM2_12";
      O;
      A     "1KM1_12";
      A     "2KM1_14";
      A     "2KM2_12";
      O;
      A     "1KM1_12";
      A     "2KM1_12";
      A     "2KM2_14";
      );
      A     "M 1.6";
      =     "M 51.2";
NETWORK
TITLE =
      A(;
      O     "M 51.0";
      O     "M 51.2";
      O     "M 51.2";
      );
      A     "M 51.4";
      =     "M 51.5";
END_FUNCTION

FUNCTION "FC 122" : VOID	// FC 122
VERSION : 0.1
BEGIN
// (block stored without names or comments; labels and parameter names are numbered)
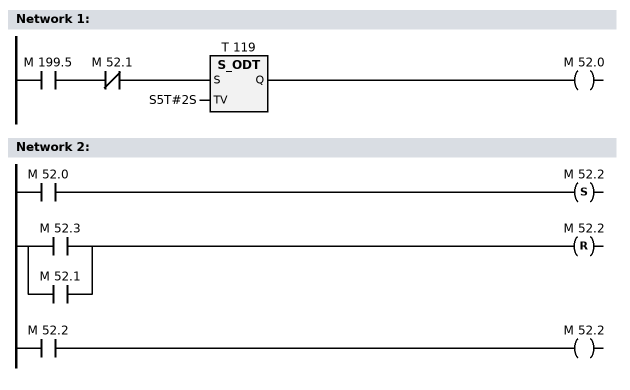
NETWORK
TITLE =
      A     "M 199.5";
      AN    "M 52.1";
      L     S5T#2S;
      SD    "T 119";
      NOP   0;
      NOP   0;
      NOP   0;
      A     "T 119";
      =     "M 52.0";
NETWORK
TITLE =
      A     "M 52.0";
      S     "M 52.2";
      A(;
      O     "M 52.3";
      O     "M 52.1";
      );
      R     "M 52.2";
      A     "M 52.2";
      =     "M 52.2";
END_FUNCTION

FUNCTION "FC 123" : VOID	// FC 123
VERSION : 0.1
BEGIN
// (block stored without names or comments; labels and parameter names are numbered)
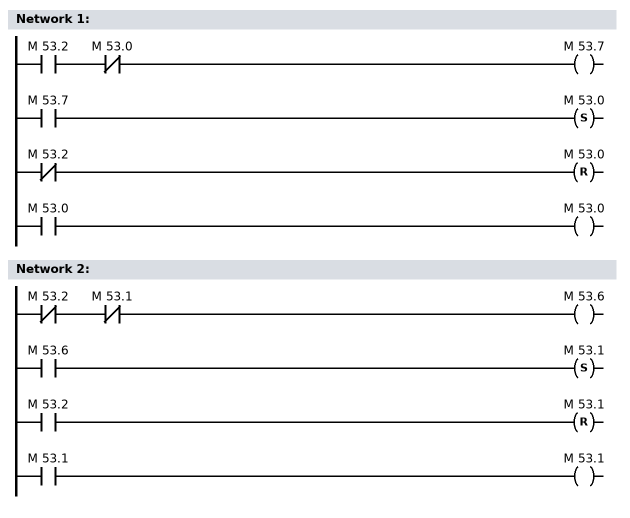
NETWORK
TITLE =
      A     "M 53.2";
      AN    "M 53.0";
      =     "M 53.7";
      A     "M 53.7";
      S     "M 53.0";
      AN    "M 53.2";
      R     "M 53.0";
      A     "M 53.0";
      =     "M 53.0";
NETWORK
TITLE =
      AN    "M 53.2";
      AN    "M 53.1";
      =     "M 53.6";
      A     "M 53.6";
      S     "M 53.1";
      A     "M 53.2";
      R     "M 53.1";
      A     "M 53.1";
      =     "M 53.1";
NETWORK
TITLE =
      A     "M 53.3";
      A     "M 53.7";
      CU    "Z 119";
      A     "M 53.3";
      A     "M 53.6";
      CD    "Z 119";
      A     "M 53.5";
      L     "MW 54";
      S     "Z 119";
      NOP   0;
      NOP   0;
      LC    "Z 119";
      T     "MW 56";
      A     "Z 119";
      =     "M 53.4";
END_FUNCTION

FUNCTION "FC 124" : VOID	// FC 124
VERSION : 0.1
BEGIN
// (block stored without names or comments; labels and parameter names are numbered)
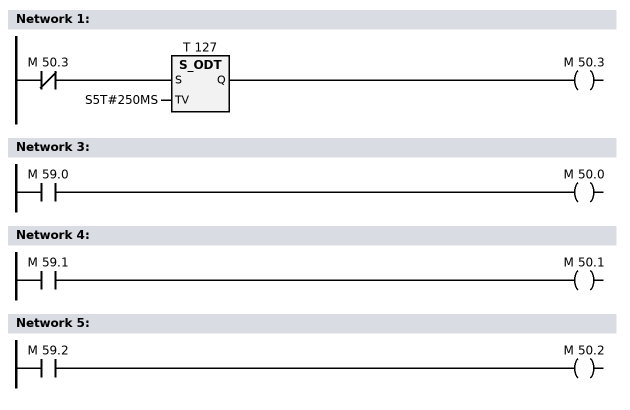
NETWORK
TITLE =
      AN    "M 50.3";
      L     S5T#250MS;
      SD    "T 127";
      NOP   0;
      NOP   0;
      NOP   0;
      A     "T 127";
      =     "M 50.3";
NETWORK
TITLE =
      A     "M 50.3";
      CU    "Z 127";
      BLD   101;
      NOP   0;
      NOP   0;
      A     "M 59.3";
      R     "Z 127";
      NOP   0;
      LC    "Z 127";
      T     "MW 58";
      NOP   0;
NETWORK
TITLE =
      A     "M 59.0";
      =     "M 50.0";
NETWORK
TITLE =
      A     "M 59.1";
      =     "M 50.1";
NETWORK
TITLE =
      A     "M 59.2";
      =     "M 50.2";
END_FUNCTION

FUNCTION "FC 125" : VOID	// FC 125
VERSION : 0.1
BEGIN
// (block stored without names or comments; labels and parameter names are numbered)
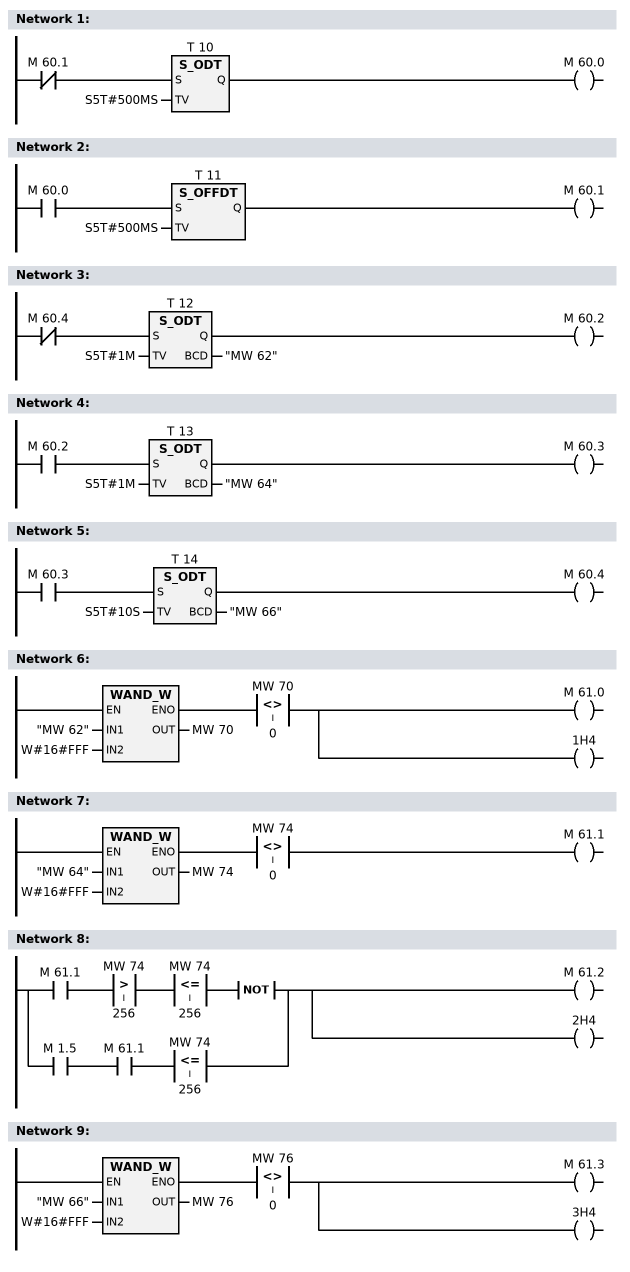
NETWORK
TITLE =
      AN    "M 60.1";
      L     S5T#500MS;
      SD    "T 10";
      NOP   0;
      NOP   0;
      NOP   0;
      A     "T 10";
      =     "M 60.0";
NETWORK
TITLE =
      A     "M 60.0";
      L     S5T#500MS;
      SF    "T 11";
      NOP   0;
      NOP   0;
      NOP   0;
      A     "T 11";
      =     "M 60.1";
NETWORK
TITLE =
      AN    "M 60.4";
      L     S5T#1M;
      SD    "T 12";
      NOP   0;
      NOP   0;
      LC    "T 12";
      T     "MW 62";
      A     "T 12";
      =     "M 60.2";
NETWORK
TITLE =
      A     "M 60.2";
      L     S5T#1M;
      SD    "T 13";
      NOP   0;
      NOP   0;
      LC    "T 13";
      T     "MW 64";
      A     "T 13";
      =     "M 60.3";
NETWORK
TITLE =
      A     "M 60.3";
      L     S5T#10S;
      SD    "T 14";
      NOP   0;
      NOP   0;
      LC    "T 14";
      T     "MW 66";
      A     "T 14";
      =     "M 60.4";
NETWORK
TITLE =
      A(;
      L     "MW 62";
      L     W#16#FFF;
      AW;
      T     MW 70;
      SET;
      SAVE;
      CLR;
      A     BR;
      );
      A(;
      L     MW 70;
      L     0;
      <>I;
      );
      =     "M 61.0";
      =     "1H4";
NETWORK
TITLE =
      A(;
      L     "MW 64";
      L     W#16#FFF;
      AW;
      T     MW 74;
      SET;
      SAVE;
      CLR;
      A     BR;
      );
      A(;
      L     MW 74;
      L     0;
      <>I;
      );
      =     "M 61.1";
NETWORK
TITLE =
      A     "M 61.1";
      A(;
      L     MW 74;
      L     256;
      >I;
      );
      A(;
      A(;
      L     MW 74;
      L     256;
      <=I;
      );
      NOT;
      );
      O;
      A     "M 1.5";
      A     "M 61.1";
      A(;
      L     MW 74;
      L     256;
      <=I;
      );
      =     "M 61.2";
      =     "2H4";
NETWORK
TITLE =
      A(;
      L     "MW 66";
      L     W#16#FFF;
      AW;
      T     MW 76;
      SET;
      SAVE;
      CLR;
      A     BR;
      );
      A(;
      L     MW 76;
      L     0;
      <>I;
      );
      =     "M 61.3";
      =     "3H4";
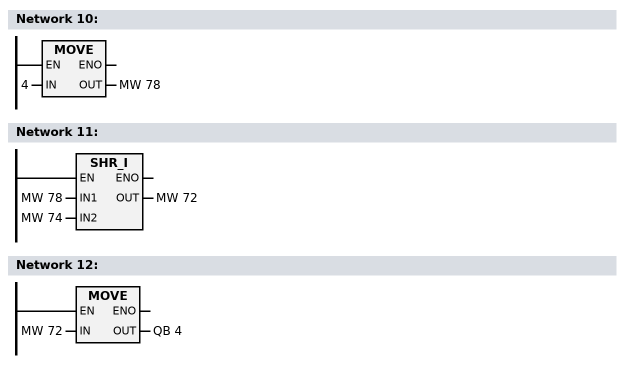
NETWORK
TITLE =
      L     4;
      T     MW 78;
      NOP   0;
NETWORK
TITLE =
      L     MW 78;
      L     MW 74;
      SSI;
      T     MW 72;
      NOP   0;
NETWORK
TITLE =
      L     MW 72;
      T     QB 4;
      NOP   0;
END_FUNCTION

FUNCTION "FC 130" : VOID	// FC 130
VERSION : 0.1
BEGIN
// (block stored without names or comments; labels and parameter names are numbered)
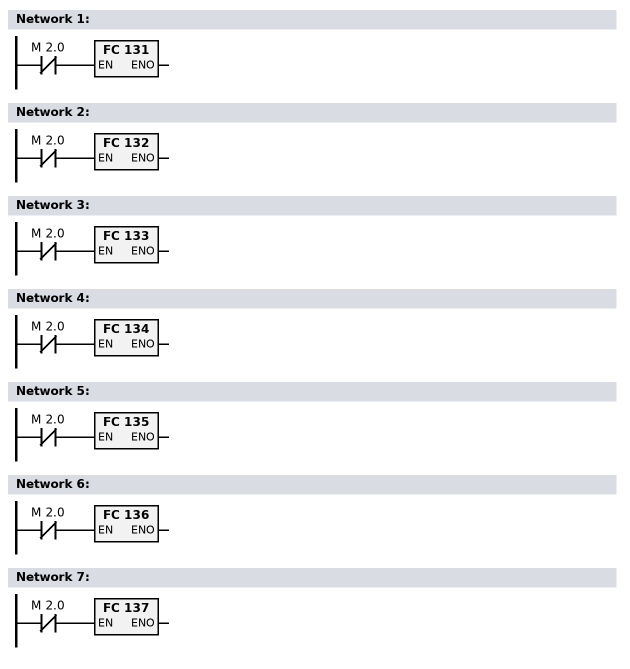
NETWORK
TITLE =
      AN    "M 2.0";
      JNB   M001;
      CALL  "FC 131";
M001: NOP   0;
NETWORK
TITLE =
      AN    "M 2.0";
      JNB   M002;
      CALL  "FC 132";
M002: NOP   0;
NETWORK
TITLE =
      AN    "M 2.0";
      JNB   M003;
      CALL  "FC 133";
M003: NOP   0;
NETWORK
TITLE =
      AN    "M 2.0";
      JNB   M004;
      CALL  "FC 134";
M004: NOP   0;
NETWORK
TITLE =
      AN    "M 2.0";
      JNB   M005;
      CALL  "FC 135";
M005: NOP   0;
NETWORK
TITLE =
      AN    "M 2.0";
      JNB   M006;
      CALL  "FC 136";
M006: NOP   0;
NETWORK
TITLE =
      AN    "M 2.0";
      JNB   M007;
      CALL  "FC 137";
M007: NOP   0;
END_FUNCTION

FUNCTION "FC 131" : VOID	// FC 131
VERSION : 0.1
BEGIN
// (block stored without names or comments; labels and parameter names are numbered)
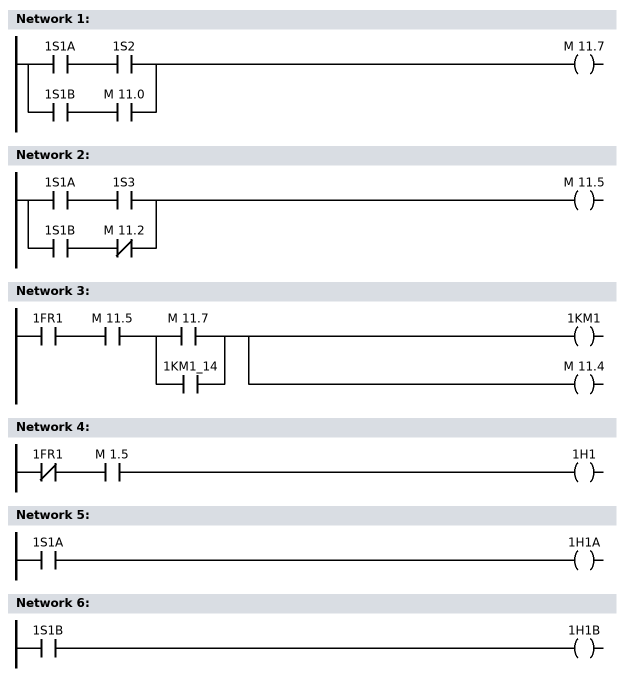
NETWORK
TITLE =
      A     "1S1A";
      A     "1S2";
      O;
      A     "1S1B";
      A     "M 11.0";
      =     "M 11.7";
NETWORK
TITLE =
      A     "1S1A";
      A     "1S3";
      O;
      A     "1S1B";
      AN    "M 11.2";
      =     "M 11.5";
NETWORK
TITLE =
      A     "1FR1";
      A     "M 11.5";
      A(;
      O     "M 11.7";
      O     "1KM1_14";
      );
      =     "1KM1";
      =     "M 11.4";
NETWORK
TITLE =
      AN    "1FR1";
      A     "M 1.5";
      =     "1H1";
NETWORK
TITLE =
      A     "1S1A";
      =     "1H1A";
NETWORK
TITLE =
      A     "1S1B";
      =     "1H1B";
END_FUNCTION

FUNCTION "FC 132" : VOID	// FC 132
VERSION : 0.1
BEGIN
// (block stored without names or comments; labels and parameter names are numbered)
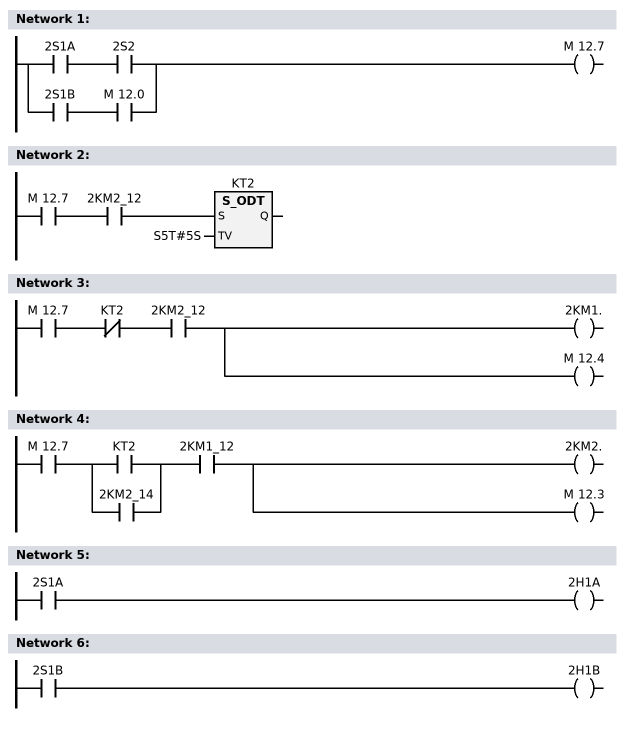
NETWORK
TITLE =
      A     "2S1A";
      A     "2S2";
      O;
      A     "2S1B";
      A     "M 12.0";
      =     "M 12.7";
NETWORK
TITLE =
      A     "M 12.7";
      A     "2KM2_12";
      L     S5T#5S;
      SD    "KT2";
      NOP   0;
      NOP   0;
      NOP   0;
      NOP   0;
NETWORK
TITLE =
      A     "M 12.7";
      AN    "KT2";
      A     "2KM2_12";
      =     "2KM1.";
      =     "M 12.4";
NETWORK
TITLE =
      A     "M 12.7";
      A(;
      O     "KT2";
      O     "2KM2_14";
      );
      A     "2KM1_12";
      =     "2KM2.";
      =     "M 12.3";
NETWORK
TITLE =
      A     "2S1A";
      =     "2H1A";
NETWORK
TITLE =
      A     "2S1B";
      =     "2H1B";
END_FUNCTION

FUNCTION "FC 133" : VOID	// FC 133
VERSION : 0.1
BEGIN
// (block stored without names or comments; labels and parameter names are numbered)
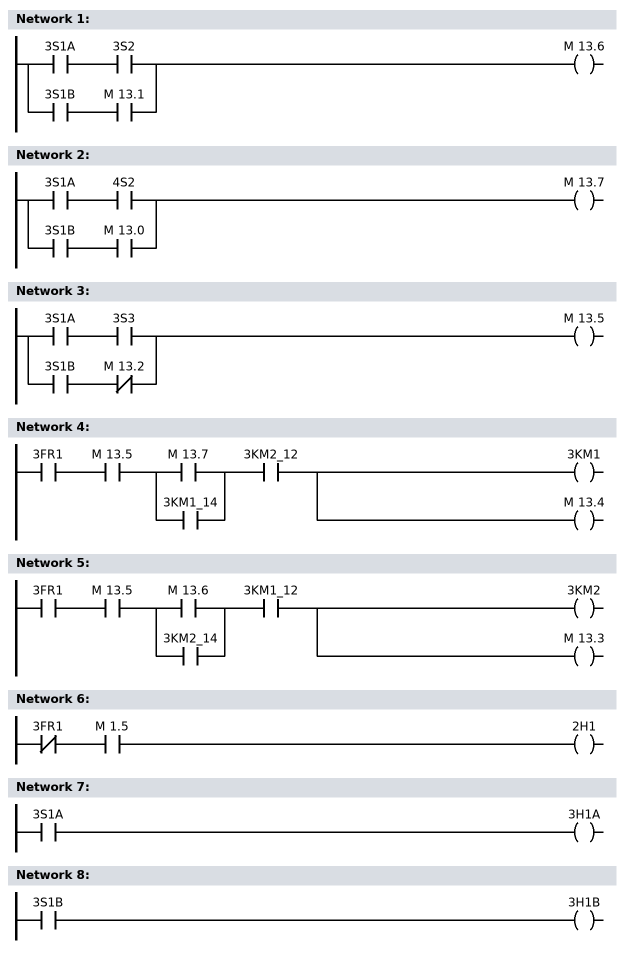
NETWORK
TITLE =
      A     "3S1A";
      A     "3S2";
      O;
      A     "3S1B";
      A     "M 13.1";
      =     "M 13.6";
NETWORK
TITLE =
      A     "3S1A";
      A     "4S2";
      O;
      A     "3S1B";
      A     "M 13.0";
      =     "M 13.7";
NETWORK
TITLE =
      A     "3S1A";
      A     "3S3";
      O;
      A     "3S1B";
      AN    "M 13.2";
      =     "M 13.5";
NETWORK
TITLE =
      A     "3FR1";
      A     "M 13.5";
      A(;
      O     "M 13.7";
      O     "3KM1_14";
      );
      A     "3KM2_12";
      =     "3KM1";
      =     "M 13.4";
NETWORK
TITLE =
      A     "3FR1";
      A     "M 13.5";
      A(;
      O     "M 13.6";
      O     "3KM2_14";
      );
      A     "3KM1_12";
      =     "3KM2";
      =     "M 13.3";
NETWORK
TITLE =
      AN    "3FR1";
      A     "M 1.5";
      =     "2H1";
NETWORK
TITLE =
      A     "3S1A";
      =     "3H1A";
NETWORK
TITLE =
      A     "3S1B";
      =     "3H1B";
END_FUNCTION

FUNCTION "FC 134" : VOID	// FC 134
VERSION : 0.1
BEGIN
// (block stored without names or comments; labels and parameter names are numbered)
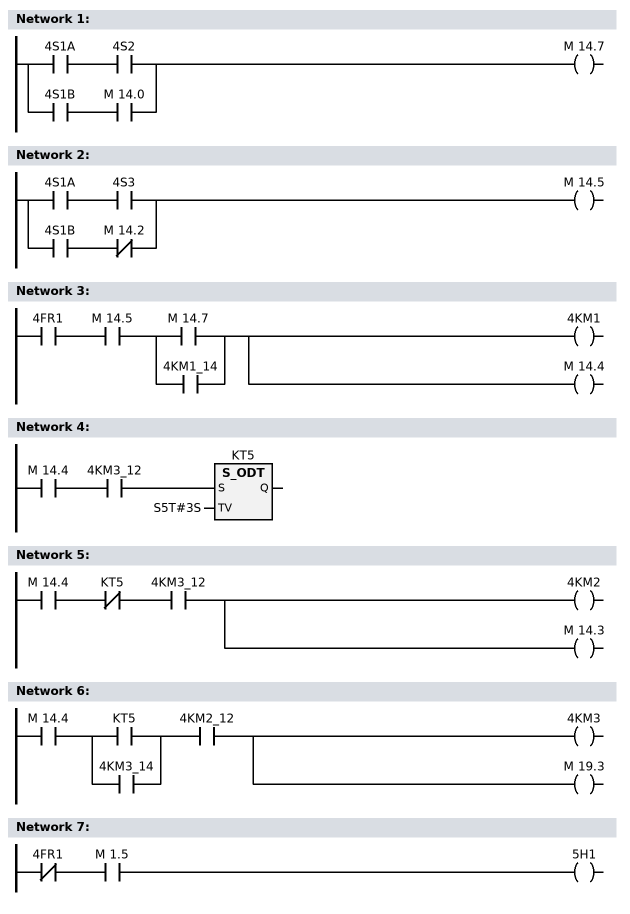
NETWORK
TITLE =
      A     "4S1A";
      A     "4S2";
      O;
      A     "4S1B";
      A     "M 14.0";
      =     "M 14.7";
NETWORK
TITLE =
      A     "4S1A";
      A     "4S3";
      O;
      A     "4S1B";
      AN    "M 14.2";
      =     "M 14.5";
NETWORK
TITLE =
      A     "4FR1";
      A     "M 14.5";
      A(;
      O     "M 14.7";
      O     "4KM1_14";
      );
      =     "4KM1";
      =     "M 14.4";
NETWORK
TITLE =
      A     "M 14.4";
      A     "4KM3_12";
      L     S5T#3S;
      SD    "KT5";
      NOP   0;
      NOP   0;
      NOP   0;
      NOP   0;
NETWORK
TITLE =
      A     "M 14.4";
      AN    "KT5";
      A     "4KM3_12";
      =     "4KM2";
      =     "M 14.3";
NETWORK
TITLE =
      A     "M 14.4";
      A(;
      O     "KT5";
      O     "4KM3_14";
      );
      A     "4KM2_12";
      =     "4KM3";
      =     "M 19.3";
NETWORK
TITLE =
      AN    "4FR1";
      A     "M 1.5";
      =     "5H1";
END_FUNCTION

FUNCTION "FC 135" : VOID	// FC 135
VERSION : 0.1
BEGIN
// (block stored without names or comments; labels and parameter names are numbered)
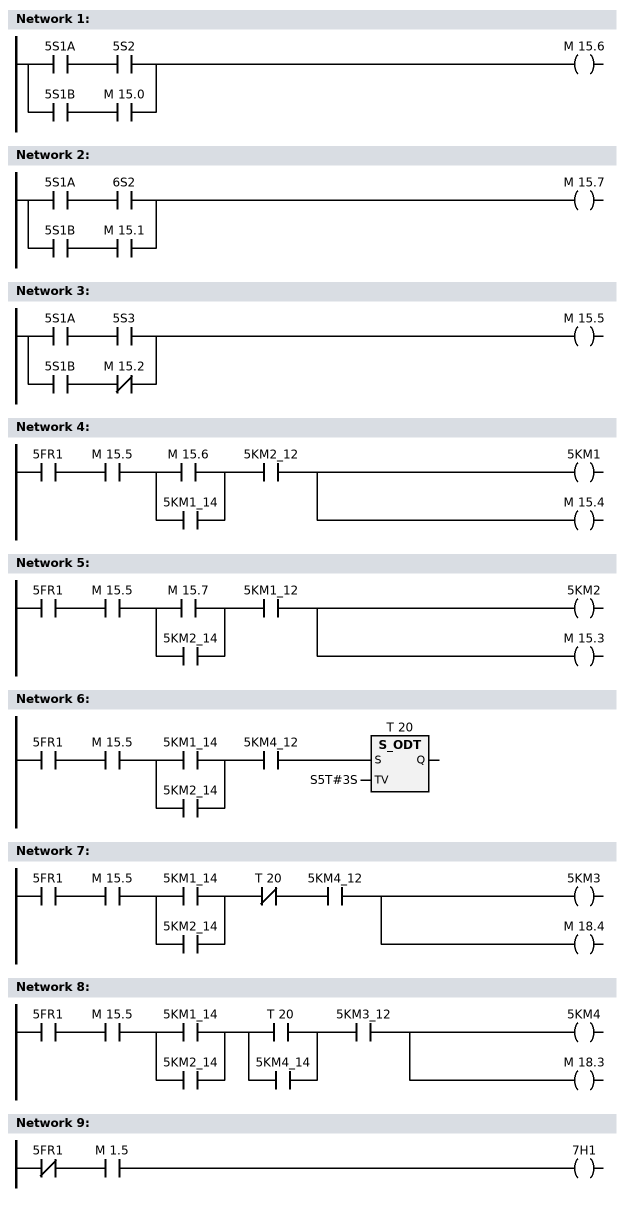
NETWORK
TITLE =
      A     "5S1A";
      A     "5S2";
      O;
      A     "5S1B";
      A     "M 15.0";
      =     "M 15.6";
NETWORK
TITLE =
      A     "5S1A";
      A     "6S2";
      O;
      A     "5S1B";
      A     "M 15.1";
      =     "M 15.7";
NETWORK
TITLE =
      A     "5S1A";
      A     "5S3";
      O;
      A     "5S1B";
      AN    "M 15.2";
      =     "M 15.5";
NETWORK
TITLE =
      A     "5FR1";
      A     "M 15.5";
      A(;
      O     "M 15.6";
      O     "5KM1_14";
      );
      A     "5KM2_12";
      =     "5KM1";
      =     "M 15.4";
NETWORK
TITLE =
      A     "5FR1";
      A     "M 15.5";
      A(;
      O     "M 15.7";
      O     "5KM2_14";
      );
      A     "5KM1_12";
      =     "5KM2";
      =     "M 15.3";
NETWORK
TITLE =
      A     "5FR1";
      A     "M 15.5";
      A(;
      O     "5KM1_14";
      O     "5KM2_14";
      );
      A     "5KM4_12";
      L     S5T#3S;
      SD    "T 20";
      NOP   0;
      NOP   0;
      NOP   0;
      NOP   0;
NETWORK
TITLE =
      A     "5FR1";
      A     "M 15.5";
      A(;
      O     "5KM1_14";
      O     "5KM2_14";
      );
      AN    "T 20";
      A     "5KM4_12";
      =     "5KM3";
      =     "M 18.4";
NETWORK
TITLE =
      A     "5FR1";
      A     "M 15.5";
      A(;
      O     "5KM1_14";
      O     "5KM2_14";
      );
      A(;
      O     "T 20";
      O     "5KM4_14";
      );
      A     "5KM3_12";
      =     "5KM4";
      =     "M 18.3";
NETWORK
TITLE =
      AN    "5FR1";
      A     "M 1.5";
      =     "7H1";
END_FUNCTION

FUNCTION "FC 136" : VOID	// FC 136
VERSION : 0.1
BEGIN
// (block stored without names or comments; labels and parameter names are numbered)
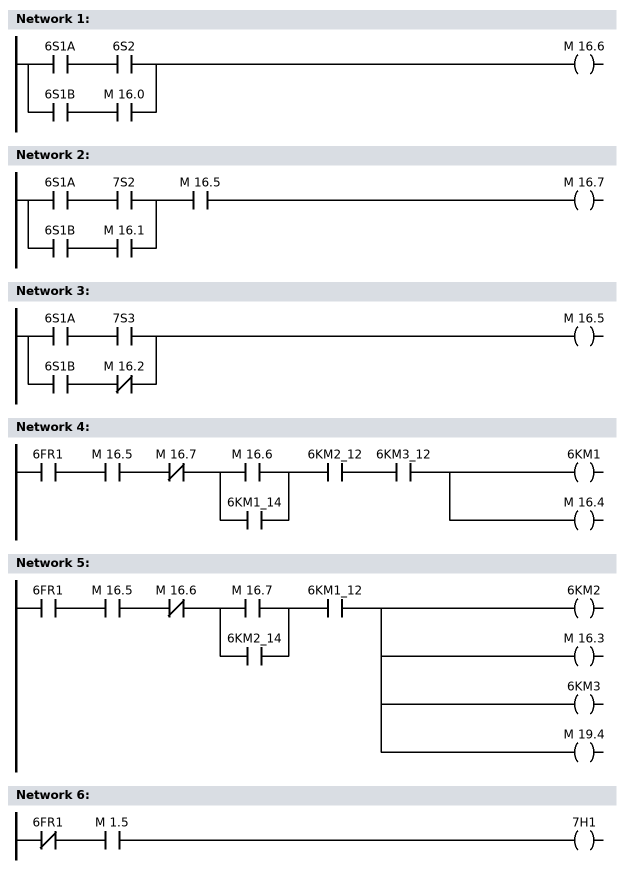
NETWORK
TITLE =
      A     "6S1A";
      A     "6S2";
      O;
      A     "6S1B";
      A     "M 16.0";
      =     "M 16.6";
NETWORK
TITLE =
      A(;
      A     "6S1A";
      A     "7S2";
      O;
      A     "6S1B";
      A     "M 16.1";
      );
      A     "M 16.5";
      =     "M 16.7";
NETWORK
TITLE =
      A     "6S1A";
      A     "7S3";
      O;
      A     "6S1B";
      AN    "M 16.2";
      =     "M 16.5";
NETWORK
TITLE =
      A     "6FR1";
      A     "M 16.5";
      AN    "M 16.7";
      A(;
      O     "M 16.6";
      O     "6KM1_14";
      );
      A     "6KM2_12";
      A     "6KM3_12";
      =     "6KM1";
      =     "M 16.4";
NETWORK
TITLE =
      A     "6FR1";
      A     "M 16.5";
      AN    "M 16.6";
      A(;
      O     "M 16.7";
      O     "6KM2_14";
      );
      A     "6KM1_12";
      =     "6KM2";
      =     "M 16.3";
      =     "6KM3";
      =     "M 19.4";
NETWORK
TITLE =
      AN    "6FR1";
      A     "M 1.5";
      =     "7H1";
END_FUNCTION

FUNCTION "FC 137" : VOID	// FC 137
VERSION : 0.1
BEGIN
// (block stored without names or comments; labels and parameter names are numbered)
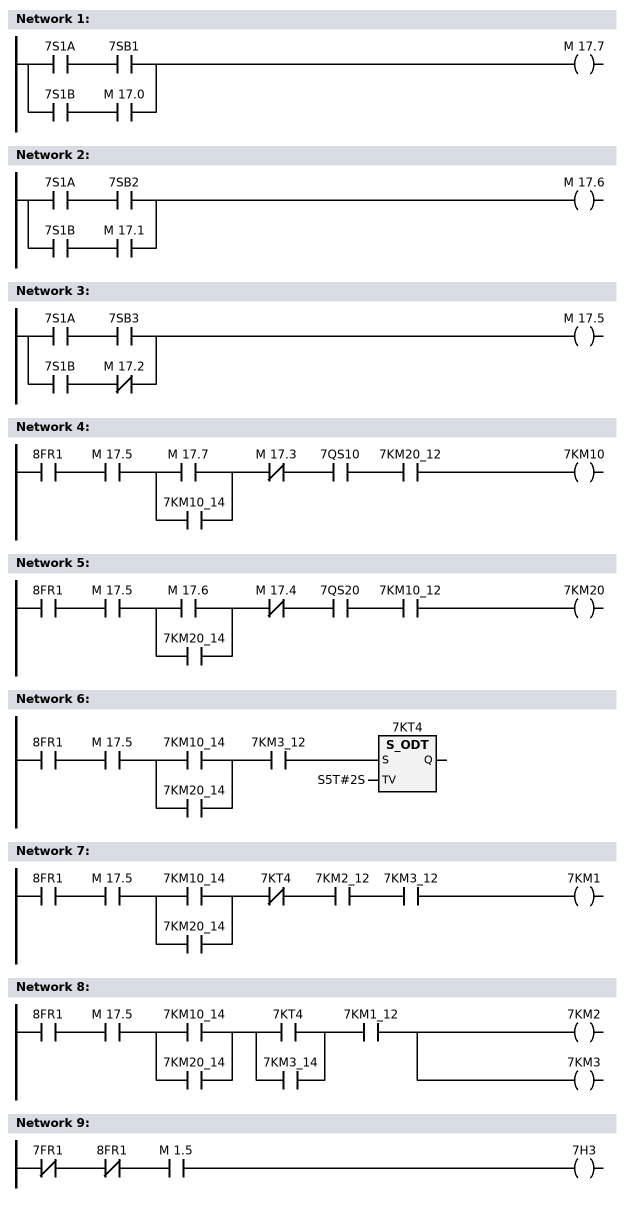
NETWORK
TITLE =
      A     "7S1A";
      A     "7SB1";
      O;
      A     "7S1B";
      A     "M 17.0";
      =     "M 17.7";
NETWORK
TITLE =
      A     "7S1A";
      A     "7SB2";
      O;
      A     "7S1B";
      A     "M 17.1";
      =     "M 17.6";
NETWORK
TITLE =
      A     "7S1A";
      A     "7SB3";
      O;
      A     "7S1B";
      AN    "M 17.2";
      =     "M 17.5";
NETWORK
TITLE =
      A     "8FR1";
      A     "M 17.5";
      A(;
      O     "M 17.7";
      O     "7KM10_14";
      );
      AN    "M 17.3";
      A     "7QS10";
      A     "7KM20_12";
      =     "7KM10";
NETWORK
TITLE =
      A     "8FR1";
      A     "M 17.5";
      A(;
      O     "M 17.6";
      O     "7KM20_14";
      );
      AN    "M 17.4";
      A     "7QS20";
      A     "7KM10_12";
      =     "7KM20";
NETWORK
TITLE =
      A     "8FR1";
      A     "M 17.5";
      A(;
      O     "7KM10_14";
      O     "7KM20_14";
      );
      A     "7KM3_12";
      L     S5T#2S;
      SD    "7KT4";
      NOP   0;
      NOP   0;
      NOP   0;
      NOP   0;
NETWORK
TITLE =
      A     "8FR1";
      A     "M 17.5";
      A(;
      O     "7KM10_14";
      O     "7KM20_14";
      );
      AN    "7KT4";
      A     "7KM2_12";
      A     "7KM3_12";
      =     "7KM1";
NETWORK
TITLE =
      A     "8FR1";
      A     "M 17.5";
      A(;
      O     "7KM10_14";
      O     "7KM20_14";
      );
      A(;
      O     "7KT4";
      O     "7KM3_14";
      );
      A     "7KM1_12";
      =     "7KM2";
      =     "7KM3";
NETWORK
TITLE =
      AN    "7FR1";
      AN    "8FR1";
      A     "M 1.5";
      =     "7H3";
END_FUNCTION

FUNCTION "FC 140" : VOID	// FC 140
VERSION : 0.1
BEGIN
// (block stored without names or comments; labels and parameter names are numbered)
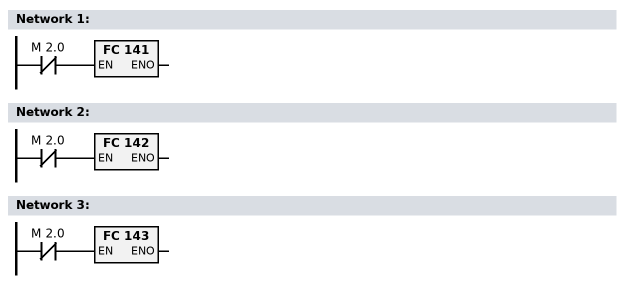
NETWORK
TITLE =
      AN    "M 2.0";
      JNB   M001;
      CALL  "FC 141";
M001: NOP   0;
NETWORK
TITLE =
      AN    "M 2.0";
      JNB   M002;
      CALL  "FC 142";
M002: NOP   0;
NETWORK
TITLE =
      AN    "M 2.0";
      JNB   M003;
      CALL  "FC 143";
M003: NOP   0;
END_FUNCTION

FUNCTION "FC 141" : VOID	// FC 141
VERSION : 0.1
BEGIN
// (block stored without names or comments; labels and parameter names are numbered)
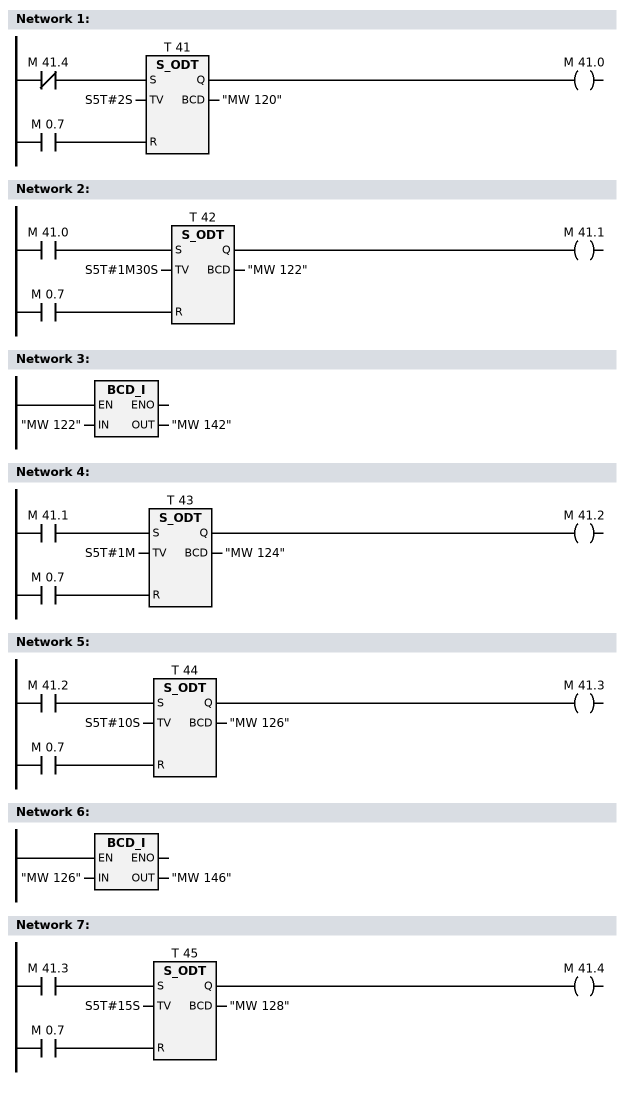
NETWORK
TITLE =
      AN    "M 41.4";
      L     S5T#2S;
      SD    "T 41";
      A     "M 0.7";
      R     "T 41";
      NOP   0;
      LC    "T 41";
      T     "MW 120";
      A     "T 41";
      =     "M 41.0";
NETWORK
TITLE =
      A     "M 41.0";
      L     S5T#1M30S;
      SD    "T 42";
      A     "M 0.7";
      R     "T 42";
      NOP   0;
      LC    "T 42";
      T     "MW 122";
      A     "T 42";
      =     "M 41.1";
NETWORK
TITLE =
      L     "MW 122";
      BTI;
      T     "MW 142";
      NOP   0;
NETWORK
TITLE =
      A     "M 41.1";
      L     S5T#1M;
      SD    "T 43";
      A     "M 0.7";
      R     "T 43";
      NOP   0;
      LC    "T 43";
      T     "MW 124";
      A     "T 43";
      =     "M 41.2";
NETWORK
TITLE =
      A     "M 41.2";
      L     S5T#10S;
      SD    "T 44";
      A     "M 0.7";
      R     "T 44";
      NOP   0;
      LC    "T 44";
      T     "MW 126";
      A     "T 44";
      =     "M 41.3";
NETWORK
TITLE =
      L     "MW 126";
      BTI;
      T     "MW 146";
      NOP   0;
NETWORK
TITLE =
      A     "M 41.3";
      L     S5T#15S;
      SD    "T 45";
      A     "M 0.7";
      R     "T 45";
      NOP   0;
      LC    "T 45";
      T     "MW 128";
      A     "T 45";
      =     "M 41.4";
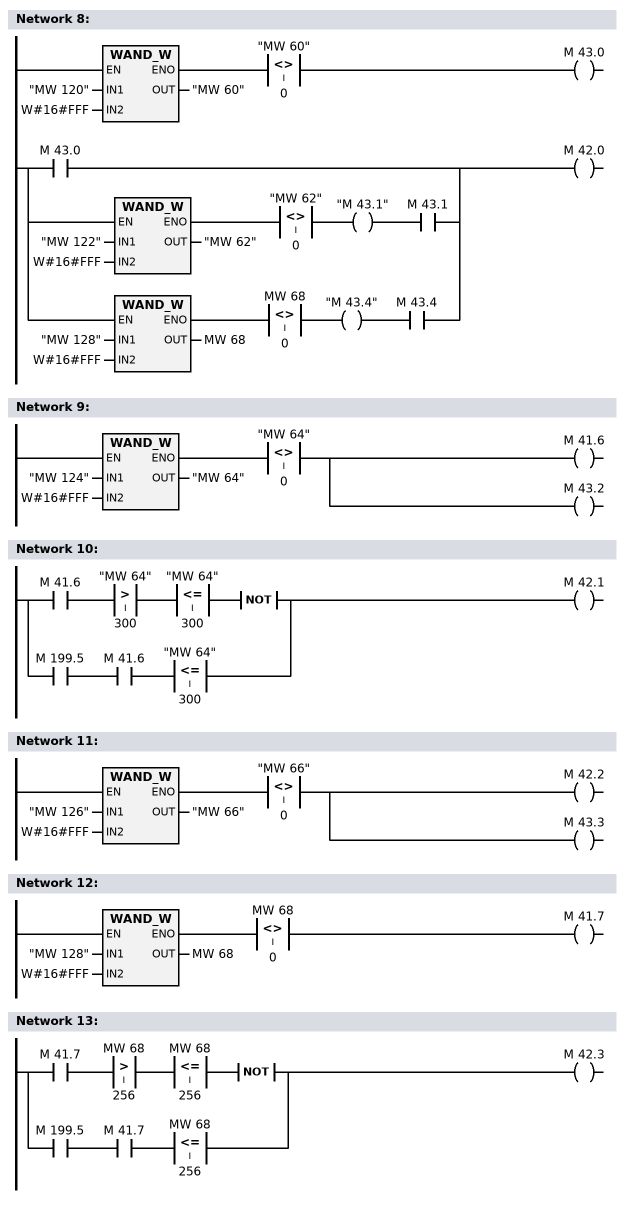
NETWORK
TITLE =
      A(;
      L     "MW 120";
      L     W#16#FFF;
      AW;
      T     "MW 60";
      SET;
      SAVE;
      CLR;
      A     BR;
      );
      A(;
      L     "MW 60";
      L     0;
      <>I;
      );
      =     "M 43.0";
      A     "M 43.0";
      O(;
      A(;
      L     "MW 122";
      L     W#16#FFF;
      AW;
      T     "MW 62";
      SET;
      SAVE;
      CLR;
      A     BR;
      );
      A(;
      L     "MW 62";
      L     0;
      <>I;
      );
      =     "M 43.1";
      A     "M 43.1";
      );
      O(;
      A(;
      L     "MW 128";
      L     W#16#FFF;
      AW;
      T     MW 68;
      SET;
      SAVE;
      CLR;
      A     BR;
      );
      A(;
      L     MW 68;
      L     0;
      <>I;
      );
      =     "M 43.4";
      A     "M 43.4";
      );
      =     "M 42.0";
NETWORK
TITLE =
      A(;
      L     "MW 124";
      L     W#16#FFF;
      AW;
      T     "MW 64";
      SET;
      SAVE;
      CLR;
      A     BR;
      );
      A(;
      L     "MW 64";
      L     0;
      <>I;
      );
      =     "M 41.6";
      =     "M 43.2";
NETWORK
TITLE =
      A     "M 41.6";
      A(;
      L     "MW 64";
      L     300;
      >I;
      );
      A(;
      A(;
      L     "MW 64";
      L     300;
      <=I;
      );
      NOT;
      );
      O;
      A     "M 199.5";
      A     "M 41.6";
      A(;
      L     "MW 64";
      L     300;
      <=I;
      );
      =     "M 42.1";
NETWORK
TITLE =
      A(;
      L     "MW 126";
      L     W#16#FFF;
      AW;
      T     "MW 66";
      SET;
      SAVE;
      CLR;
      A     BR;
      );
      A(;
      L     "MW 66";
      L     0;
      <>I;
      );
      =     "M 42.2";
      =     "M 43.3";
NETWORK
TITLE =
      A(;
      L     "MW 128";
      L     W#16#FFF;
      AW;
      T     MW 68;
      SET;
      SAVE;
      CLR;
      A     BR;
      );
      A(;
      L     MW 68;
      L     0;
      <>I;
      );
      =     "M 41.7";
NETWORK
TITLE =
      A     "M 41.7";
      A(;
      L     MW 68;
      L     256;
      >I;
      );
      A(;
      A(;
      L     MW 68;
      L     256;
      <=I;
      );
      NOT;
      );
      O;
      A     "M 199.5";
      A     "M 41.7";
      A(;
      L     MW 68;
      L     256;
      <=I;
      );
      =     "M 42.3";
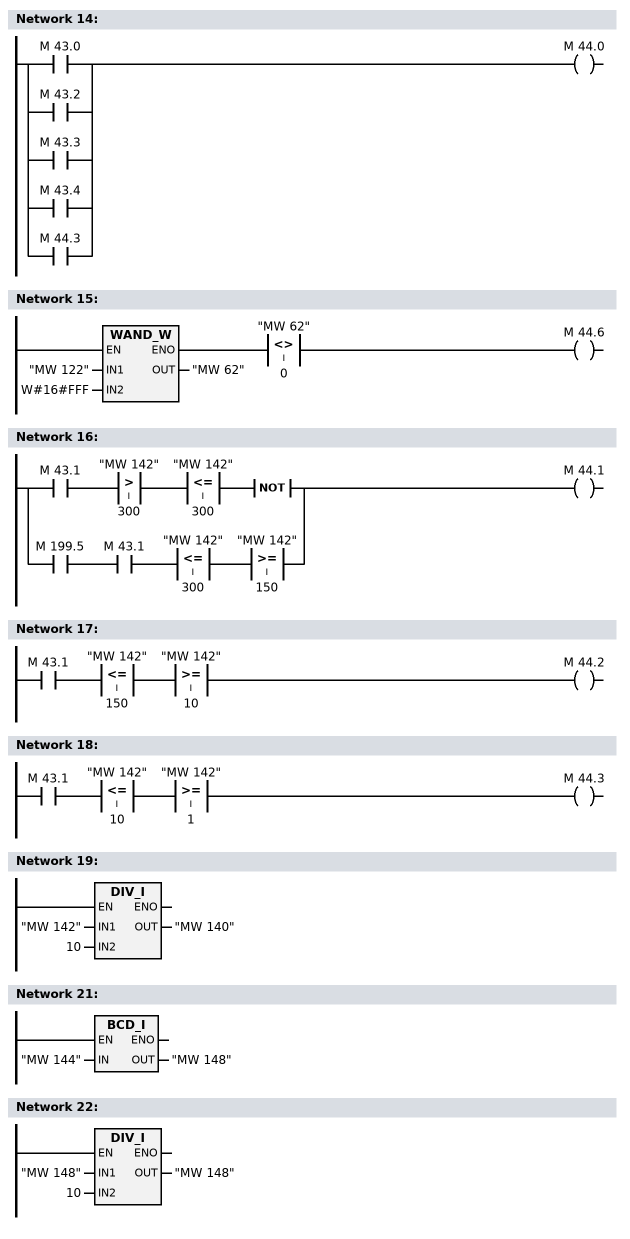
NETWORK
TITLE =
      O     "M 43.0";
      O     "M 43.2";
      O     "M 43.3";
      O     "M 43.4";
      O     M 44.3;
      =     "M 44.0";
NETWORK
TITLE =
      A(;
      L     "MW 122";
      L     W#16#FFF;
      AW;
      T     "MW 62";
      SET;
      SAVE;
      CLR;
      A     BR;
      );
      A(;
      L     "MW 62";
      L     0;
      <>I;
      );
      =     "M 44.6";
NETWORK
TITLE =
      A     "M 43.1";
      A(;
      L     "MW 142";
      L     300;
      >I;
      );
      A(;
      A(;
      L     "MW 142";
      L     300;
      <=I;
      );
      NOT;
      );
      O;
      A     "M 199.5";
      A     "M 43.1";
      A(;
      L     "MW 142";
      L     300;
      <=I;
      );
      A(;
      L     "MW 142";
      L     150;
      >=I;
      );
      =     "M 44.1";
NETWORK
TITLE =
      A     "M 43.1";
      A(;
      L     "MW 142";
      L     150;
      <=I;
      );
      A(;
      L     "MW 142";
      L     10;
      >=I;
      );
      =     "M 44.2";
NETWORK
TITLE =
      A     "M 43.1";
      A(;
      L     "MW 142";
      L     10;
      <=I;
      );
      A(;
      L     "MW 142";
      L     1;
      >=I;
      );
      =     M 44.3;
NETWORK
TITLE =
      L     "MW 142";
      L     10;
      /I;
      T     "MW 140";
      NOP   0;
NETWORK
TITLE =
      A(;
      A     "M 44.0";
      S     M 43.7;
      A     M 44.3;
      R     M 43.7;
      A     M 43.7;
      );
      L     S5T#1M10S;
      SD    "T 46";
      NOP   0;
      NOP   0;
      LC    "T 46";
      T     "MW 144";
      NOP   0;
NETWORK
TITLE =
      L     "MW 144";
      BTI;
      T     "MW 148";
      NOP   0;
NETWORK
TITLE =
      L     "MW 148";
      L     10;
      /I;
      T     "MW 148";
      NOP   0;
END_FUNCTION

FUNCTION "FC 142" : VOID	// FC 142
VERSION : 0.1
BEGIN
// (block stored without names or comments; labels and parameter names are numbered)
NETWORK
TITLE =
      A     "M 139.0";
      A     "M 139.1";
      CU    "Z 100";
      BLD   101;
      NOP   0;
      NOP   0;
      A(;
      L     "MW 150";
      L     60;
      >=I;
      );
      R     "Z 100";
      NOP   0;
      LC    "Z 100";
      T     "MW 160";
      NOP   0;
